C08961=1010.506,304.090,-163.238,-18.890,47.066,37.479
C08962=1010.613,303.852,-163.048,-19.485,46.587,36.235
C08963=1010.718,303.613,-162.860,-20.052,46.107,35.019
C08964=1010.823,303.374,-162.672,-20.593,45.627,33.826
C08965=1010.904,303.186,-162.527,-20.997,45.253,32.914
C08966=1010.984,302.998,-162.383,-21.384,44.880,32.017
C08967=1011.063,302.809,-162.239,-21.757,44.508,31.133
C08968=1011.142,302.619,-162.097,-22.115,44.137,30.264
C08969=1011.243,302.376,-161.916,-22.552,43.665,29.173
C08970=1011.342,302.132,-161.736,-22.967,43.196,28.105
C08971=1011.440,301.887,-161.558,-23.359,42.732,27.060
C08972=1011.536,301.641,-161.381,-23.731,42.271,26.037
C08973=1011.612,301.446,-161.243,-24.011,41.910,25.243
C08974=1011.687,301.252,-161.105,-24.278,41.553,24.463
C08975=1011.761,301.056,-160.968,-24.533,41.199,23.695
C08976=1011.835,300.859,-160.832,-24.778,40.847,22.938
C08977=1011.928,300.610,-160.662,-25.071,40.409,21.999
C08978=1012.020,300.361,-160.491,-25.349,39.974,21.077
C08979=1012.110,300.110,-160.323,-25.611,39.544,20.170
///RCONF 0,0,0,0,1,0,0,0,0,0,0,0,0,0,0,0,0,0,0,0,0,0,0,0
C08980=1012.200,299.859,-160.157,-25.857,39.121,19.283
C08981=1012.270,299.658,-160.024,-26.044,38.787,18.584
C08982=1012.340,299.456,-159.894,-26.221,38.458,17.898
C08983=1012.410,299.255,-159.763,-26.391,38.132,17.220
C08984=1012.478,299.051,-159.633,-26.551,37.810,16.553
C08985=1012.564,298.798,-159.472,-26.741,37.414,15.733
C08986=1012.647,298.543,-159.313,-26.918,37.024,14.926
C08987=1012.731,298.287,-159.155,-27.085,36.640,14.133
C08988=1012.814,298.031,-158.998,-27.241,36.263,13.354
C08989=1012.880,297.824,-158.872,-27.359,35.964,12.737
C08990=1012.944,297.618,-158.747,-27.470,35.670,12.129
C08991=1013.009,297.410,-158.624,-27.576,35.380,11.529
C08992=1013.072,297.202,-158.500,-27.675,35.094,10.935
C08993=1013.151,296.943,-158.349,-27.790,34.746,10.213
C08994=1013.228,296.685,-158.199,-27.897,34.404,9.500
C08995=1013.305,296.425,-158.050,-27.996,34.069,8.801
C08996=1013.380,296.164,-157.902,-28.087,33.740,8.111
C08997=1013.441,295.953,-157.783,-28.156,33.478,7.560
C08998=1013.502,295.741,-157.665,-28.220,33.220,7.016
C08999=1013.561,295.528,-157.547,-28.280,32.966,6.479
C09000=1013.621,295.315,-157.430,-28.335,32.716,5.947
C09001=1013.692,295.052,-157.288,-28.398,32.417,5.306
C09002=1013.763,294.790,-157.147,-28.455,32.123,4.674
C09003=1013.833,294.526,-157.006,-28.506,31.835,4.050
C09004=1013.902,294.263,-156.867,-28.552,31.552,3.436
C09005=1013.958,294.047,-156.754,-28.586,31.327,2.940
C09006=1014.014,293.830,-156.642,-28.617,31.104,2.450
C09007=1014.070,293.613,-156.531,-28.645,30.886,1.967
C09008=1014.124,293.395,-156.420,-28.669,30.673,1.490
C09009=1014.190,293.130,-156.286,-28.695,30.417,0.916
C09010=1014.254,292.865,-156.154,-28.717,30.168,0.353
C09011=1014.318,292.598,-156.022,-28.736,29.926,-0.203
C09012=1014.382,292.331,-155.891,-28.751,29.686,-0.753
C09013=1014.434,292.111,-155.784,-28.760,29.494,-1.200
C09014=1014.485,291.891,-155.678,-28.768,29.306,-1.642
C09015=1014.535,291.669,-155.572,-28.773,29.120,-2.080
C09016=1014.586,291.448,-155.467,-28.777,28.937,-2.514
C09017=1014.646,291.180,-155.341,-28.778,28.722,-3.030
C09018=1014.705,290.912,-155.217,-28.777,28.512,-3.541
C09019=1014.763,290.643,-155.093,-28.773,28.305,-4.046
C09020=1014.821,290.373,-154.970,-28.767,28.103,-4.544
C09021=1014.869,290.149,-154.869,-28.760,27.939,-4.952
C09022=1014.915,289.926,-154.768,-28.752,27.779,-5.357
C09023=1014.962,289.701,-154.668,-28.742,27.622,-5.757
C09024=1015.008,289.476,-154.569,-28.730,27.467,-6.153
C09025=1015.063,289.207,-154.450,-28.715,27.285,-6.624
C09026=1015.116,288.935,-154.333,-28.698,27.109,-7.088
C09027=1015.170,288.665,-154.217,-28.679,26.937,-7.545
C09028=1015.222,288.394,-154.102,-28.659,26.767,-7.999
C09029=1015.266,288.166,-154.006,-28.641,26.630,-8.372
C09030=1015.309,287.939,-153.911,-28.622,26.495,-8.743
C09031=1015.351,287.712,-153.816,-28.602,26.363,-9.109
C09032=1015.393,287.483,-153.722,-28.581,26.233,-9.471
C09033=1015.442,287.211,-153.611,-28.555,26.082,-9.899
C09034=1015.492,286.940,-153.500,-28.527,25.936,-10.320
C09035=1015.540,286.667,-153.391,-28.499,25.792,-10.737
C09036=1015.587,286.394,-153.283,-28.470,25.652,-11.148
C09037=1015.627,286.164,-153.192,-28.444,25.537,-11.492
C09038=1015.665,285.933,-153.102,-28.418,25.425,-11.832
C09039=1015.705,285.704,-153.012,-28.391,25.314,-12.171
C09040=1015.743,285.473,-152.924,-28.364,25.204,-12.507
C09041=1015.787,285.199,-152.820,-28.330,25.079,-12.901
C09042=1015.832,284.926,-152.716,-28.296,24.955,-13.292
C09043=1015.875,284.652,-152.614,-28.261,24.835,-13.680
C09044=1015.918,284.378,-152.512,-28.226,24.716,-14.065
C09045=1015.954,284.145,-152.426,-28.195,24.619,-14.388
C09046=1015.989,283.912,-152.341,-28.164,24.524,-14.708
C09047=1016.024,283.680,-152.256,-28.132,24.429,-15.026
C09048=1016.059,283.447,-152.172,-28.100,24.338,-15.343
C09049=1016.099,283.173,-152.075,-28.062,24.232,-15.713
C09050=1016.138,282.897,-151.978,-28.023,24.128,-16.079
C09051=1016.177,282.623,-151.881,-27.984,24.027,-16.441
C09052=1016.216,282.348,-151.786,-27.945,23.929,-16.801
C09053=1016.248,282.113,-151.705,-27.911,23.848,-17.104
C09054=1016.280,281.878,-151.625,-27.877,23.768,-17.406
C09055=1016.311,281.643,-151.545,-27.842,23.690,-17.706
C09056=1016.343,281.407,-151.466,-27.807,23.613,-18.004
C09057=1016.378,281.132,-151.374,-27.766,23.526,-18.349
C09058=1016.414,280.857,-151.284,-27.725,23.440,-18.691
C09059=1016.448,280.581,-151.193,-27.684,23.357,-19.031
C09060=1016.482,280.304,-151.104,-27.642,23.276,-19.367
C09061=1016.511,280.068,-151.028,-27.606,23.208,-19.653
C09062=1016.539,279.830,-150.952,-27.570,23.142,-19.936
C09063=1016.567,279.594,-150.877,-27.534,23.078,-20.218
C09064=1016.595,279.357,-150.803,-27.498,23.014,-20.499
C09065=1016.626,279.080,-150.717,-27.456,22.942,-20.824
C09066=1016.658,278.804,-150.632,-27.413,22.873,-21.147
C09067=1016.689,278.527,-150.548,-27.370,22.804,-21.469
C09068=1016.718,278.250,-150.465,-27.327,22.737,-21.789
C09069=1016.743,278.012,-150.393,-27.290,22.681,-22.062
C09070=1016.769,277.773,-150.322,-27.252,22.626,-22.334
C09071=1016.793,277.535,-150.252,-27.215,22.573,-22.606
C09072=1016.818,277.296,-150.183,-27.177,22.521,-22.877
C09073=1016.846,277.019,-150.102,-27.134,22.462,-23.186
C09074=1016.872,276.741,-150.023,-27.090,22.404,-23.496
C09075=1016.899,276.464,-149.944,-27.046,22.349,-23.804
C09076=1016.925,276.187,-149.866,-27.003,22.294,-24.111
C09077=1016.947,275.947,-149.800,-26.965,22.250,-24.373
C09078=1016.969,275.706,-149.733,-26.927,22.204,-24.635
C09079=1016.990,275.466,-149.667,-26.889,22.162,-24.896
C09080=1017.012,275.226,-149.602,-26.851,22.119,-25.156
C09081=1017.035,274.949,-149.528,-26.807,22.073,-25.453
C09082=1017.058,274.670,-149.454,-26.763,22.027,-25.750
C09083=1017.080,274.393,-149.380,-26.720,21.983,-26.043
C09084=1017.103,274.115,-149.308,-26.676,21.940,-26.336
C09085=1017.122,273.874,-149.246,-26.638,21.903,-26.590
C09086=1017.140,273.632,-149.184,-26.600,21.869,-26.841
C09087=1017.158,273.391,-149.123,-26.562,21.835,-27.092
C09088=1017.176,273.149,-149.062,-26.525,21.803,-27.342
C09089=1017.197,272.871,-148.993,-26.481,21.766,-27.626
C09090=1017.216,272.593,-148.925,-26.438,21.731,-27.910
C09091=1017.234,272.315,-148.857,-26.395,21.697,-28.194
C09092=1017.254,272.036,-148.790,-26.351,21.664,-28.476
C09093=1017.269,271.793,-148.732,-26.314,21.637,-28.720
C09094=1017.284,271.550,-148.675,-26.276,21.610,-28.964
C09095=1017.299,271.308,-148.618,-26.238,21.585,-29.208
C09096=1017.315,271.065,-148.561,-26.201,21.560,-29.450
C09097=1017.330,270.786,-148.498,-26.158,21.533,-29.728
C09098=1017.346,270.508,-148.435,-26.115,21.507,-30.003
C09099=1017.361,270.229,-148.372,-26.072,21.483,-30.277
C09100=1017.376,269.951,-148.310,-26.030,21.459,-30.551
C09101=1017.388,269.707,-148.257,-25.992,21.439,-30.791
C09102=1017.400,269.462,-148.204,-25.955,21.420,-31.029
C09103=1017.413,269.219,-148.151,-25.918,21.402,-31.266
C09104=1017.424,268.974,-148.098,-25.881,21.386,-31.502
C09105=1017.436,268.696,-148.040,-25.839,21.367,-31.772
C09106=1017.449,268.417,-147.983,-25.797,21.350,-32.039
C09107=1017.461,268.139,-147.926,-25.755,21.333,-32.307
C09108=1017.472,267.860,-147.869,-25.713,21.318,-32.573
C09109=1017.481,267.616,-147.820,-25.677,21.306,-32.805
C09110=1017.490,267.370,-147.771,-25.641,21.295,-33.037
C09111=1017.499,267.125,-147.723,-25.604,21.284,-33.269
C09112=1017.508,266.879,-147.676,-25.568,21.275,-33.499
C09113=1017.516,266.601,-147.622,-25.527,21.264,-33.760
C09114=1017.525,266.322,-147.569,-25.487,21.254,-34.021
C09115=1017.533,266.043,-147.517,-25.446,21.246,-34.279
C09116=1017.540,265.765,-147.465,-25.406,21.239,-34.538
C09117=1017.547,265.519,-147.421,-25.370,21.233,-34.766
C09118=1017.553,265.273,-147.376,-25.335,21.229,-34.991
C09119=1017.559,265.026,-147.333,-25.300,21.225,-35.219
C09120=1017.564,264.780,-147.290,-25.265,21.221,-35.444
C09121=1017.570,264.501,-147.242,-25.226,21.219,-35.699
C09122=1017.574,264.222,-147.194,-25.186,21.217,-35.952
C09123=1017.579,263.943,-147.146,-25.147,21.216,-36.205
C09124=1017.584,263.664,-147.100,-25.108,21.215,-36.458
C09125=1017.586,263.417,-147.059,-25.074,21.216,-36.681
C09126=1017.590,263.170,-147.020,-25.040,21.217,-36.903
C09127=1017.592,262.923,-146.980,-25.006,21.220,-37.124
C09128=1017.594,262.676,-146.941,-24.973,21.223,-37.345
C09129=1017.597,262.397,-146.898,-24.935,21.227,-37.593
C09130=1017.598,262.117,-146.855,-24.897,21.233,-37.842
C09131=1017.600,261.839,-146.813,-24.860,21.238,-38.090
C09132=1017.600,261.559,-146.771,-24.823,21.245,-38.337
C09133=1017.601,261.311,-146.736,-24.790,21.251,-38.554
C09134=1017.601,261.064,-146.700,-24.758,21.259,-38.770
C09135=1017.600,260.816,-146.665,-24.725,21.267,-38.988
C09136=1017.599,260.568,-146.631,-24.693,21.275,-39.204
C09137=1017.598,260.289,-146.592,-24.658,21.287,-39.446
C09138=1017.596,260.009,-146.554,-24.622,21.298,-39.688
C09139=1017.594,259.730,-146.517,-24.587,21.310,-39.930
C09140=1017.592,259.450,-146.481,-24.551,21.322,-40.171
C09141=1017.575,258.214,-146.327,-24.430,21.375,-41.012
C09142=1017.571,257.971,-146.298,-24.430,21.375,-41.014
C09143=1017.568,257.727,-146.269,-24.429,21.375,-41.018
C09144=1017.565,257.483,-146.240,-24.429,21.376,-41.019
C09145=1017.560,257.241,-146.210,-24.429,21.376,-41.021
C09146=1017.557,256.997,-146.181,-24.428,21.375,-41.025
C09147=1017.554,256.754,-146.152,-24.428,21.376,-41.027
C09148=1017.551,256.510,-146.123,-24.428,21.377,-41.029
C09149=1017.548,256.262,-146.094,-24.427,21.376,-41.032
C09150=1017.544,256.014,-146.063,-24.427,21.376,-41.034
C09151=1017.541,255.766,-146.035,-24.426,21.376,-41.037
C09152=1017.537,255.518,-146.005,-24.426,21.377,-41.040
C09153=1017.534,255.269,-145.975,-24.426,21.377,-41.042
C09154=1017.530,255.021,-145.945,-24.425,21.377,-41.045
C09155=1017.527,254.772,-145.916,-24.425,21.377,-41.047
C09156=1017.524,254.524,-145.887,-24.425,21.377,-41.049
C09157=1017.520,254.276,-145.856,-24.424,21.378,-41.052
C09158=1017.517,254.028,-145.828,-24.424,21.378,-41.054
C09159=1017.514,253.780,-145.797,-24.424,21.378,-41.058
C09160=1017.510,253.532,-145.768,-24.423,21.378,-41.060
C09161=1017.508,253.283,-145.739,-24.423,21.378,-41.061
C09162=1017.504,253.035,-145.709,-24.423,21.378,-41.065
C09163=1017.501,252.787,-145.680,-24.422,21.379,-41.067
C09164=1017.497,252.538,-145.651,-24.422,21.379,-41.069
C09165=1017.494,252.291,-145.621,-24.421,21.378,-41.072
C09166=1017.491,252.042,-145.591,-24.421,21.379,-41.074
C09167=1017.488,251.794,-145.562,-24.421,21.380,-41.076
C09168=1017.484,251.545,-145.533,-24.421,21.380,-41.078
C09169=1017.482,251.302,-145.504,-24.420,21.380,-41.082
C09170=1017.478,251.059,-145.475,-24.420,21.380,-41.084
C09171=1017.475,250.815,-145.446,-24.420,21.380,-41.085
C09172=1017.472,250.572,-145.417,-24.419,21.380,-41.089
C09173=1017.468,250.329,-145.389,-24.419,21.380,-41.091
C09174=1017.466,250.086,-145.360,-24.419,21.381,-41.093
C09175=1017.462,249.842,-145.332,-24.418,21.381,-41.095
C09176=1017.459,249.598,-145.303,-24.418,21.381,-41.098
C09177=1017.456,249.350,-145.274,-24.418,21.381,-41.100
C09178=1017.453,249.102,-145.244,-24.417,21.381,-41.102
C09179=1017.449,248.853,-145.215,-24.417,21.381,-41.104
C09180=1017.447,248.606,-145.185,-24.417,21.381,-41.107
C09181=1017.443,248.358,-145.156,-24.416,21.381,-41.109
C09182=1017.440,248.109,-145.127,-24.416,21.382,-41.111
C09183=1017.437,247.861,-145.098,-24.416,21.382,-41.113
C09184=1017.434,247.613,-145.069,-24.415,21.382,-41.117
C09185=1017.430,247.364,-145.039,-24.415,21.382,-41.118
C09186=1017.427,247.116,-145.011,-24.415,21.382,-41.120
C09187=1017.425,246.868,-144.981,-24.414,21.383,-41.122
C09188=1017.421,246.620,-144.952,-24.414,21.382,-41.126
C09189=1017.419,246.371,-144.923,-24.414,21.382,-41.127
C09190=1017.415,246.123,-144.894,-24.413,21.383,-41.129
C09191=1017.413,245.875,-144.865,-24.413,21.384,-41.132
C09192=1017.409,245.627,-144.836,-24.413,21.384,-41.134
C09193=1017.406,245.379,-144.807,-24.412,21.384,-41.137
C09194=1017.403,245.130,-144.777,-24.412,21.384,-41.139
C09195=1017.400,244.882,-144.748,-24.412,21.384,-41.141
C09196=1017.397,244.633,-144.719,-24.412,21.384,-41.143
C09197=1017.394,244.390,-144.692,-24.411,21.384,-41.144
C09198=1017.391,244.146,-144.662,-24.411,21.384,-41.148
C09199=1017.388,243.904,-144.634,-24.411,21.384,-41.150
C09200=1017.385,243.660,-144.606,-24.410,21.384,-41.151
C09201=1017.382,243.418,-144.578,-24.410,21.385,-41.153
C09202=1017.379,243.173,-144.549,-24.410,21.385,-41.155
C09203=1017.376,242.931,-144.521,-24.410,21.385,-41.157
C09204=1017.374,242.688,-144.492,-24.409,21.385,-41.159
C09205=1017.370,242.440,-144.463,-24.409,21.385,-41.162
C09206=1017.367,242.191,-144.435,-24.408,21.385,-41.164
C09207=1017.364,241.942,-144.405,-24.408,21.385,-41.166
C09208=1017.361,241.694,-144.377,-24.408,21.386,-41.168
C09209=1017.358,241.446,-144.347,-24.408,21.386,-41.170
C09210=1017.355,241.198,-144.319,-24.407,21.386,-41.172
C09211=1017.353,240.949,-144.290,-24.407,21.386,-41.174
C09212=1017.350,240.701,-144.261,-24.407,21.386,-41.177
C09213=1017.346,240.453,-144.232,-24.406,21.386,-41.179
C09214=1017.344,240.204,-144.204,-24.406,21.386,-41.181
C09215=1017.341,239.956,-144.175,-24.406,21.386,-41.183
C09216=1017.338,239.708,-144.145,-24.406,21.387,-41.184
C09217=1017.335,239.460,-144.117,-24.405,21.387,-41.186
C09218=1017.332,239.212,-144.089,-24.405,21.387,-41.188
C09219=1017.330,238.963,-144.059,-24.405,21.387,-41.190
C09220=1017.327,238.715,-144.031,-24.405,21.388,-41.192
C09221=1017.324,238.466,-144.002,-24.404,21.387,-41.195
C09222=1017.321,238.218,-143.974,-24.404,21.387,-41.197
C09223=1017.318,237.970,-143.945,-24.403,21.388,-41.199
C09224=1017.315,237.722,-143.916,-24.403,21.388,-41.201
C09225=1017.312,237.478,-143.888,-24.403,21.388,-41.203
C09226=1017.310,237.235,-143.859,-24.403,21.388,-41.205
C09227=1017.307,236.992,-143.832,-24.402,21.388,-41.207
C09228=1017.305,236.749,-143.803,-24.402,21.389,-41.209
C09229=1017.301,236.506,-143.775,-24.402,21.389,-41.210
C09230=1017.299,236.263,-143.748,-24.402,21.389,-41.212
C09231=1017.296,236.019,-143.719,-24.401,21.389,-41.214
C09232=1017.293,235.777,-143.691,-24.401,21.390,-41.216
C09233=1017.291,235.528,-143.662,-24.401,21.389,-41.218
C09234=1017.288,235.280,-143.634,-24.401,21.389,-41.219
C09235=1017.285,235.031,-143.606,-24.400,21.389,-41.221
C09236=1017.283,234.784,-143.577,-24.400,21.390,-41.223
C09237=1017.280,234.535,-143.549,-24.400,21.390,-41.225
C09238=1017.277,234.287,-143.519,-24.400,21.390,-41.227
C09239=1017.274,234.038,-143.491,-24.399,21.390,-41.229
C09240=1017.271,233.790,-143.463,-24.399,21.390,-41.231
C09241=1017.269,233.541,-143.434,-24.399,21.391,-41.233
C09242=1017.266,233.293,-143.406,-24.399,21.391,-41.234
C09243=1017.264,233.045,-143.377,-24.398,21.391,-41.236
C09244=1017.261,232.797,-143.349,-24.398,21.390,-41.238
C09245=1017.258,232.548,-143.320,-24.398,21.391,-41.240
C09246=1017.255,232.300,-143.291,-24.397,21.391,-41.242
C09247=1017.252,232.051,-143.263,-24.397,21.391,-41.243
C09248=1017.249,231.803,-143.234,-24.397,21.391,-41.245
C09249=1017.248,231.555,-143.206,-24.397,21.392,-41.247
C09250=1017.245,231.306,-143.178,-24.396,21.392,-41.249
C09251=1017.242,231.057,-143.149,-24.396,21.392,-41.251
C09252=1017.239,230.809,-143.120,-24.396,21.391,-41.252
C09253=1017.237,230.587,-143.095,-24.396,21.392,-41.254
C09254=1017.235,230.365,-143.071,-24.395,21.392,-41.256
C09255=1017.233,230.143,-143.045,-24.395,21.392,-41.258
C09256=1017.230,229.920,-143.020,-24.395,21.392,-41.258
C09257=1017.228,229.698,-142.994,-24.395,21.392,-41.260
C09258=1017.225,229.476,-142.969,-24.395,21.392,-41.262
C09259=1017.223,229.254,-142.943,-24.394,21.393,-41.264
C09260=1017.221,229.031,-142.917,-24.394,21.392,-41.265
C09261=1017.218,228.783,-142.889,-24.394,21.392,-41.267
C09262=1017.216,228.535,-142.862,-24.394,21.392,-41.269
C09263=1017.214,228.286,-142.833,-24.393,21.393,-41.271
C09264=1017.210,228.038,-142.804,-24.393,21.393,-41.273
C09265=1017.209,227.790,-142.776,-24.393,21.394,-41.273
C09266=1017.206,227.541,-142.748,-24.393,21.393,-41.275
C09267=1017.203,227.292,-142.720,-24.393,21.393,-41.276
C09268=1017.201,227.044,-142.691,-24.392,21.394,-41.278
C09269=1017.198,226.796,-142.663,-24.392,21.394,-41.280
C09270=1017.195,226.548,-142.635,-24.392,21.394,-41.282
C09271=1017.193,226.299,-142.606,-24.392,21.394,-41.284
C09272=1017.190,226.051,-142.578,-24.391,21.394,-41.285
C09273=1017.188,225.802,-142.550,-24.391,21.394,-41.287
C09274=1017.186,225.554,-142.522,-24.391,21.394,-41.289
C09275=1017.183,225.305,-142.494,-24.390,21.394,-41.291
C09276=1017.181,225.057,-142.465,-24.391,21.395,-41.291
C09277=1017.179,224.767,-142.433,-24.390,21.395,-41.293
C09278=1017.176,224.478,-142.400,-24.390,21.395,-41.295
C09279=1017.172,224.188,-142.367,-24.389,21.394,-41.298
C09280=1017.169,223.898,-142.335,-24.389,21.395,-41.300
C09281=1017.167,223.655,-142.306,-24.389,21.395,-41.300
C09282=1017.165,223.412,-142.279,-24.389,21.396,-41.302
C09283=1017.162,223.170,-142.252,-24.389,21.396,-41.304
C09284=1017.160,222.926,-142.224,-24.388,21.395,-41.306
C09285=1017.158,222.684,-142.197,-24.388,21.395,-41.308
C09286=1017.155,222.441,-142.170,-24.388,21.396,-41.309
C09287=1017.153,222.198,-142.141,-24.388,21.397,-41.310
C09288=1017.151,221.955,-142.114,-24.388,21.396,-41.311
C09289=1017.148,221.706,-142.086,-24.387,21.396,-41.313
C09290=1017.146,221.458,-142.058,-24.387,21.396,-41.315
C09291=1017.143,221.210,-142.030,-24.387,21.397,-41.317
C09292=1017.141,220.961,-142.003,-24.386,21.396,-41.318
C09293=1017.139,220.712,-141.974,-24.386,21.396,-41.320
C09294=1017.137,220.464,-141.946,-24.386,21.397,-41.321
C09295=1017.134,220.216,-141.918,-24.386,21.397,-41.323
C09296=1017.132,219.968,-141.890,-24.386,21.397,-41.324
C09297=1017.130,219.720,-141.862,-24.385,21.397,-41.326
C09298=1017.128,219.471,-141.834,-24.385,21.397,-41.328
C09299=1017.125,219.222,-141.807,-24.385,21.397,-41.330
C09300=1017.123,218.974,-141.779,-24.385,21.397,-41.330
C09301=1017.121,218.725,-141.750,-24.385,21.397,-41.332
C09302=1017.118,218.477,-141.722,-24.384,21.398,-41.333
C09303=1017.116,218.229,-141.695,-24.384,21.398,-41.335
C09304=1017.114,217.980,-141.667,-24.384,21.397,-41.337
C09305=1017.111,217.732,-141.639,-24.384,21.397,-41.339
C09306=1017.110,217.483,-141.611,-24.384,21.398,-41.339
C09307=1017.107,217.236,-141.583,-24.383,21.399,-41.341
C09308=1017.105,216.986,-141.556,-24.383,21.398,-41.342
C09309=1017.102,216.744,-141.528,-24.383,21.398,-41.344
C09310=1017.101,216.501,-141.501,-24.383,21.398,-41.346
C09311=1017.098,216.258,-141.473,-24.383,21.398,-41.346
C09312=1017.096,216.015,-141.447,-24.382,21.399,-41.348
C09313=1017.094,215.773,-141.420,-24.382,21.399,-41.350
C09314=1017.092,215.530,-141.392,-24.382,21.399,-41.352
C09315=1017.090,215.287,-141.365,-24.382,21.398,-41.353
C09316=1017.088,215.045,-141.338,-24.382,21.399,-41.354
C09317=1017.086,214.795,-141.310,-24.381,21.400,-41.356
C09318=1017.083,214.547,-141.282,-24.381,21.399,-41.357
C09319=1017.081,214.299,-141.255,-24.381,21.399,-41.359
C09320=1017.080,214.051,-141.227,-24.381,21.400,-41.359
C09321=1017.077,213.802,-141.199,-24.381,21.400,-41.361
C09322=1017.075,213.554,-141.172,-24.380,21.400,-41.363
C09323=1017.073,213.305,-141.143,-24.380,21.400,-41.365
C09324=1017.071,213.057,-141.116,-24.380,21.400,-41.366
C09325=1017.069,212.808,-141.088,-24.380,21.400,-41.366
C09326=1017.066,212.560,-141.060,-24.380,21.400,-41.368
C09327=1017.064,212.312,-141.033,-24.379,21.400,-41.370
C09328=1017.063,212.063,-141.005,-24.379,21.400,-41.372
C09329=1017.060,211.814,-140.977,-24.379,21.401,-41.372
C09330=1017.058,211.566,-140.950,-24.379,21.401,-41.374
C09331=1017.056,211.318,-140.922,-24.378,21.400,-41.375
C09332=1017.054,211.070,-140.894,-24.378,21.400,-41.377
C09333=1017.052,210.820,-140.866,-24.378,21.401,-41.378
C09334=1017.050,210.572,-140.839,-24.378,21.401,-41.379
C09335=1017.048,210.324,-140.812,-24.378,21.401,-41.381
C09336=1017.046,210.076,-140.783,-24.377,21.401,-41.383
C09337=1017.044,209.832,-140.757,-24.377,21.401,-41.383
C09338=1017.042,209.590,-140.730,-24.377,21.401,-41.385
C09339=1017.040,209.348,-140.703,-24.377,21.402,-41.387
C09340=1017.038,209.105,-140.677,-24.377,21.401,-41.388
C09341=1017.036,208.862,-140.649,-24.377,21.402,-41.389
C09342=1017.034,208.619,-140.622,-24.376,21.402,-41.391
C09343=1017.032,208.377,-140.595,-24.376,21.401,-41.392
C09344=1017.030,208.134,-140.569,-24.376,21.402,-41.392
C09345=1017.029,207.886,-140.541,-24.376,21.402,-41.394
C09346=1017.027,207.637,-140.514,-24.376,21.402,-41.396
C09347=1017.024,207.389,-140.486,-24.375,21.402,-41.398
C09348=1017.022,207.140,-140.458,-24.375,21.402,-41.398
C09349=1017.020,206.891,-140.431,-24.375,21.402,-41.399
C09350=1017.019,206.643,-140.403,-24.375,21.402,-41.401
C09351=1017.017,206.395,-140.376,-24.375,21.402,-41.401
C09352=1017.015,206.146,-140.349,-24.375,21.403,-41.403
C09353=1017.013,205.898,-140.321,-24.374,21.403,-41.405
C09354=1017.011,205.649,-140.294,-24.374,21.402,-41.407
C09355=1017.009,205.401,-140.267,-24.374,21.403,-41.407
C09356=1017.007,205.153,-140.238,-24.374,21.403,-41.409
C09357=1017.005,204.904,-140.211,-24.373,21.403,-41.410
C09358=1017.004,204.655,-140.184,-24.374,21.404,-41.411
C09359=1017.002,204.407,-140.157,-24.373,21.403,-41.412
C09360=1017.000,204.159,-140.129,-24.373,21.403,-41.414
C09361=1016.998,203.910,-140.101,-24.373,21.404,-41.415
C09362=1016.996,203.662,-140.074,-24.373,21.403,-41.416
C09363=1016.990,202.446,-139.939,-24.425,21.378,-41.051
C09364=1016.989,202.057,-139.895,-24.424,21.378,-41.052
C09365=1016.989,201.709,-139.856,-24.424,21.378,-41.054
C09366=1016.989,201.358,-139.818,-24.424,21.378,-41.058
C09367=1016.990,200.950,-139.773,-24.423,21.379,-41.060
C09368=1016.991,200.722,-139.748,-24.423,21.378,-41.061
C09369=1016.991,200.494,-139.723,-24.423,21.378,-41.063
C09370=1016.991,200.271,-139.699,-24.423,21.378,-41.065
C09371=1016.992,200.058,-139.675,-24.423,21.378,-41.065
C09372=1016.992,199.658,-139.631,-24.422,21.379,-41.069
C09373=1016.992,199.269,-139.589,-24.422,21.379,-41.071
C09374=1016.994,198.870,-139.545,-24.421,21.379,-41.074
C09375=1016.994,198.469,-139.502,-24.421,21.379,-41.076
C09376=1016.995,198.068,-139.458,-24.421,21.380,-41.078
C09377=1016.995,197.666,-139.414,-24.420,21.380,-41.082
C09378=1016.996,197.266,-139.369,-24.420,21.380,-41.084
C09379=1016.997,196.864,-139.326,-24.419,21.380,-41.087
C09380=1016.998,196.463,-139.283,-24.419,21.380,-41.089
C09381=1016.998,196.062,-139.239,-24.419,21.381,-41.091
C09382=1016.999,195.661,-139.195,-24.418,21.380,-41.094
C09383=1017.000,195.260,-139.151,-24.418,21.381,-41.097
C09384=1017.001,194.859,-139.107,-24.418,21.381,-41.100
C09385=1017.002,194.458,-139.064,-24.417,21.381,-41.102
C09386=1017.002,194.057,-139.021,-24.417,21.381,-41.105
C09387=1017.003,193.656,-138.977,-24.417,21.382,-41.108
C09388=1017.004,193.255,-138.933,-24.416,21.382,-41.109
C09389=1017.005,192.853,-138.889,-24.416,21.382,-41.113
C09390=1017.006,192.452,-138.846,-24.415,21.382,-41.115
C09391=1017.006,192.051,-138.803,-24.415,21.382,-41.118
C09392=1017.007,191.650,-138.760,-24.415,21.382,-41.120
C09393=1017.008,191.249,-138.716,-24.414,21.382,-41.124
C09394=1017.009,190.848,-138.672,-24.414,21.383,-41.126
C09395=1017.010,190.446,-138.628,-24.414,21.383,-41.128
C09396=1017.011,190.046,-138.585,-24.413,21.383,-41.131
C09397=1017.012,189.645,-138.542,-24.413,21.383,-41.133
C09398=1017.013,189.243,-138.499,-24.412,21.384,-41.137
C09399=1017.013,188.842,-138.455,-24.412,21.384,-41.139
C09400=1017.014,188.441,-138.412,-24.412,21.384,-41.141
C09401=1017.016,188.041,-138.369,-24.411,21.384,-41.144
C09402=1017.016,187.639,-138.326,-24.411,21.385,-41.146
C09403=1017.018,187.238,-138.282,-24.411,21.384,-41.150
C09404=1017.019,186.837,-138.239,-24.410,21.384,-41.151
C09405=1017.020,186.436,-138.196,-24.410,21.384,-41.155
C09406=1017.021,186.035,-138.152,-24.410,21.385,-41.157
C09407=1017.022,185.634,-138.109,-24.409,21.385,-41.159
C09408=1017.023,185.233,-138.066,-24.409,21.385,-41.162
C09409=1017.024,184.832,-138.023,-24.409,21.386,-41.165
C09410=1017.025,184.431,-137.980,-24.408,21.386,-41.168
C09411=1017.026,184.030,-137.936,-24.408,21.386,-41.170
C09412=1017.027,183.630,-137.894,-24.407,21.386,-41.172
C09413=1017.028,183.228,-137.850,-24.407,21.386,-41.176
C09414=1017.029,182.828,-137.807,-24.407,21.387,-41.177
C09415=1017.030,182.426,-137.765,-24.406,21.386,-41.181
C09416=1017.031,182.026,-137.722,-24.406,21.387,-41.183
C09417=1017.032,181.624,-137.678,-24.405,21.387,-41.186
C09418=1017.034,181.224,-137.635,-24.405,21.387,-41.188
C09419=1017.034,180.824,-137.593,-24.405,21.387,-41.190
C09420=1017.035,180.422,-137.551,-24.404,21.388,-41.194
C09421=1017.037,180.021,-137.508,-24.404,21.388,-41.196
C09422=1017.038,179.621,-137.465,-24.403,21.388,-41.199
C09423=1017.039,179.220,-137.421,-24.403,21.388,-41.201
C09424=1017.040,178.819,-137.378,-24.403,21.388,-41.205
C09425=1017.042,178.418,-137.336,-24.402,21.388,-41.207
C09426=1017.042,178.017,-137.293,-24.402,21.389,-41.209
C09427=1017.044,177.616,-137.250,-24.402,21.389,-41.212
C09428=1017.044,177.216,-137.208,-24.401,21.389,-41.214
C09429=1017.046,176.815,-137.165,-24.401,21.389,-41.218
C09430=1017.047,176.414,-137.122,-24.401,21.389,-41.219
C09431=1017.048,176.013,-137.079,-24.400,21.390,-41.223
C09432=1017.050,175.612,-137.037,-24.400,21.390,-41.225
C09433=1017.050,175.212,-136.994,-24.400,21.390,-41.227
C09434=1017.052,174.811,-136.951,-24.399,21.390,-41.231
C09435=1017.053,174.410,-136.909,-24.399,21.391,-41.233
C09436=1017.055,174.010,-136.866,-24.398,21.390,-41.236
C09437=1017.055,173.610,-136.824,-24.398,21.390,-41.238
C09438=1017.057,173.208,-136.782,-24.397,21.391,-41.242
C09439=1017.058,172.808,-136.739,-24.397,21.391,-41.243
C09440=1017.060,172.407,-136.696,-24.397,21.391,-41.247
C09441=1017.061,172.007,-136.654,-24.396,21.392,-41.249
C09442=1017.062,171.606,-136.611,-24.396,21.392,-41.251
C09443=1017.064,171.205,-136.569,-24.396,21.392,-41.254
C09444=1017.064,170.805,-136.527,-24.395,21.392,-41.256
C09445=1017.066,170.405,-136.484,-24.395,21.392,-41.260
C09446=1017.068,170.004,-136.442,-24.395,21.392,-41.262
C09447=1017.068,169.604,-136.399,-24.394,21.392,-41.265
C09448=1017.070,169.203,-136.357,-24.394,21.393,-41.267
C09449=1017.071,168.802,-136.315,-24.393,21.393,-41.271
C09450=1017.073,168.403,-136.272,-24.393,21.393,-41.273
C09451=1017.074,168.001,-136.230,-24.393,21.394,-41.275
C09452=1017.075,167.601,-136.188,-24.392,21.394,-41.278
C09453=1017.077,167.200,-136.146,-24.392,21.394,-41.280
C09454=1017.078,166.801,-136.104,-24.391,21.393,-41.284
C09455=1017.079,166.400,-136.061,-24.391,21.395,-41.286
C09456=1017.081,166.000,-136.019,-24.391,21.394,-41.289
C09457=1017.082,165.599,-135.977,-24.390,21.394,-41.291
C09458=1017.083,165.199,-135.935,-24.390,21.395,-41.295
C09459=1017.085,164.798,-135.893,-24.390,21.395,-41.297
C09460=1017.086,164.398,-135.850,-24.389,21.395,-41.300
C09461=1017.088,164.012,-135.811,-24.389,21.395,-41.302
C09462=1017.088,163.822,-135.790,-24.389,21.395,-41.304
C09463=1017.089,163.410,-135.747,-24.388,21.396,-41.306
C09464=1017.090,163.175,-135.722,-24.388,21.395,-41.308
C09465=1017.091,162.921,-135.696,-24.388,21.396,-41.309
C09466=1017.092,162.658,-135.667,-24.388,21.396,-41.311
C09467=1017.093,162.389,-135.640,-24.387,21.396,-41.313
C09468=1017.094,162.118,-135.611,-24.387,21.396,-41.315
C09469=1017.095,161.849,-135.583,-24.387,21.397,-41.317
C09470=1017.096,161.585,-135.556,-24.387,21.397,-41.319
C09471=1017.097,161.336,-135.529,-24.386,21.396,-41.320
C09472=1017.098,161.098,-135.504,-24.386,21.396,-41.322
C09473=1017.098,160.873,-135.481,-24.386,21.397,-41.324
C09474=1017.099,160.661,-135.459,-24.386,21.397,-41.325
C09475=1017.101,160.255,-135.416,-24.385,21.397,-41.328
C09476=1017.102,159.858,-135.374,-24.385,21.397,-41.330
C09477=1017.106,159.457,-135.334,-24.384,21.398,-41.333
C09478=1017.112,159.058,-135.295,-24.384,21.398,-41.335
C09479=1017.119,158.656,-135.256,-24.384,21.397,-41.339
C09480=1017.126,158.254,-135.218,-24.383,21.399,-41.341
C09481=1017.132,157.851,-135.179,-24.383,21.398,-41.344
C09482=1017.138,157.448,-135.140,-24.383,21.398,-41.346
C09483=1017.145,157.043,-135.101,-24.382,21.399,-41.350
C09484=1017.152,156.639,-135.062,-24.382,21.399,-41.352
C09485=1017.158,156.232,-135.023,-24.381,21.399,-41.355
C09486=1017.165,155.826,-134.983,-24.381,21.400,-41.358
C09487=1017.172,155.419,-134.944,-24.381,21.399,-41.361
C09488=1017.178,155.009,-134.905,-24.380,21.400,-41.363
C09489=1017.185,154.601,-134.865,-24.380,21.400,-41.366
C09490=1017.191,154.191,-134.826,-24.380,21.400,-41.368
C09491=1017.197,153.780,-134.786,-24.379,21.401,-41.372
C09492=1017.204,153.369,-134.746,-24.378,21.400,-41.375
C09493=1017.210,152.957,-134.707,-24.378,21.400,-41.377
C09494=1017.217,152.545,-134.666,-24.378,21.401,-41.381
C09495=1017.224,152.132,-134.628,-24.377,21.401,-41.383
C09496=1017.230,151.720,-134.587,-24.377,21.402,-41.387
C09497=1017.236,151.306,-134.547,-24.377,21.402,-41.389
C09498=1017.243,150.893,-134.508,-24.376,21.401,-41.392
C09499=1017.249,150.478,-134.467,-24.376,21.402,-41.394
C09500=1017.256,150.065,-134.427,-24.375,21.402,-41.398
C09501=1017.263,149.651,-134.388,-24.375,21.402,-41.401
C09502=1017.268,149.236,-134.348,-24.375,21.403,-41.403
C09503=1017.275,148.823,-134.308,-24.374,21.403,-41.407
C09504=1017.281,148.409,-134.268,-24.374,21.403,-41.409
C09505=1017.287,147.995,-134.228,-24.373,21.403,-41.412
C09506=1017.293,147.580,-134.189,-24.373,21.403,-41.416
C09507=1017.300,147.167,-134.149,-24.372,21.404,-41.418
C09508=1017.306,146.754,-134.109,-24.372,21.404,-41.422
C09509=1017.313,146.340,-134.069,-24.372,21.404,-41.424
C09510=1017.318,145.927,-134.030,-24.371,21.405,-41.427
C09511=1017.325,145.515,-133.990,-24.371,21.404,-41.431
C09512=1017.331,145.103,-133.950,-24.370,21.405,-41.432
C09513=1017.337,144.692,-133.910,-24.370,21.405,-41.436
C09514=1017.343,144.280,-133.870,-24.370,21.405,-41.438
C09515=1017.349,143.871,-133.831,-24.369,21.406,-41.442
C09516=1017.355,143.461,-133.792,-24.369,21.405,-41.445
C09517=1017.361,143.053,-133.753,-24.368,21.406,-41.448
C09518=1017.367,142.644,-133.713,-24.368,21.406,-41.451
C09519=1017.373,142.237,-133.674,-24.368,21.406,-41.453
C09520=1017.379,141.831,-133.635,-24.367,21.407,-41.457
C09521=1017.385,141.426,-133.596,-24.366,21.406,-41.460
C09522=1017.391,141.021,-133.557,-24.366,21.407,-41.462
C09523=1017.397,140.604,-133.517,-24.366,21.408,-41.466
C09524=1017.400,140.368,-133.495,-24.366,21.408,-41.468
C09525=1017.404,140.109,-133.470,-24.365,21.408,-41.470
C09526=1017.408,139.832,-133.443,-24.365,21.408,-41.471
C09527=1017.412,139.544,-133.416,-24.365,21.408,-41.473
C09528=1017.416,139.256,-133.388,-24.364,21.408,-41.475
C09529=1017.420,138.979,-133.361,-24.364,21.407,-41.476
C09530=1017.423,138.719,-133.337,-24.364,21.408,-41.478
C09531=1017.427,138.482,-133.314,-24.364,21.408,-41.480
C09532=1017.430,138.265,-133.293,-24.363,21.408,-41.482
C09533=1017.433,138.059,-133.273,-24.363,21.408,-41.484
C09534=1017.439,137.658,-133.234,-24.363,21.408,-41.486
C09535=1017.445,137.288,-133.199,-24.363,21.410,-41.488
C09536=1017.449,136.951,-133.167,-24.362,21.409,-41.491
C09537=1017.453,136.635,-133.136,-24.361,21.409,-41.495
C09538=1017.458,136.317,-133.106,-24.361,21.410,-41.497
C09539=1017.462,135.978,-133.073,-24.361,21.409,-41.500
C09540=1017.468,135.606,-133.038,-24.360,21.410,-41.502
C09541=1017.473,135.211,-133.000,-24.360,21.411,-41.505
C09542=1017.478,134.812,-132.962,-24.360,21.410,-41.508
C09543=1017.484,134.414,-132.923,-24.359,21.411,-41.510
C09544=1017.490,134.014,-132.885,-24.359,21.411,-41.514
C09545=1017.495,133.617,-132.847,-24.358,21.411,-41.517
C09546=1017.500,133.217,-132.809,-24.358,21.412,-41.519
C09547=1017.506,132.819,-132.771,-24.358,21.411,-41.523
C09548=1017.511,132.420,-132.732,-24.357,21.412,-41.525
C09549=1017.517,132.021,-132.695,-24.357,21.412,-41.528
C09550=1017.522,131.623,-132.656,-24.356,21.412,-41.532
C09551=1017.528,131.224,-132.618,-24.356,21.413,-41.534
C09552=1017.533,130.825,-132.580,-24.356,21.413,-41.538
C09553=1017.539,130.427,-132.542,-24.355,21.413,-41.541
C09554=1017.543,130.028,-132.504,-24.355,21.413,-41.543
C09555=1017.549,129.629,-132.466,-24.354,21.413,-41.547
C09556=1017.554,129.231,-132.427,-24.354,21.413,-41.550
C09557=1017.560,128.832,-132.390,-24.354,21.414,-41.552
C09558=1017.565,128.434,-132.351,-24.353,21.414,-41.555
C09559=1017.570,128.036,-132.313,-24.353,21.415,-41.558
C09560=1017.575,127.636,-132.275,-24.352,21.414,-41.561
C09561=1017.581,127.239,-132.237,-24.352,21.415,-41.565
C09562=1017.585,126.839,-132.199,-24.351,21.415,-41.567
C09563=1017.591,126.441,-132.160,-24.351,21.415,-41.571
C09564=1017.596,126.042,-132.123,-24.350,21.415,-41.574
C09565=1017.601,125.644,-132.085,-24.350,21.416,-41.576
C09566=1017.607,125.245,-132.047,-24.350,21.416,-41.580
C09567=1017.611,124.846,-132.008,-24.349,21.416,-41.583
C09568=1017.617,124.448,-131.971,-24.349,21.416,-41.585
C09569=1017.621,124.049,-131.933,-24.348,21.417,-41.589
C09570=1017.627,123.651,-131.895,-24.348,21.416,-41.592
C09571=1017.632,123.252,-131.856,-24.348,21.418,-41.595
C09572=1017.636,122.854,-131.818,-24.347,21.417,-41.598
C09573=1017.642,122.455,-131.781,-24.347,21.418,-41.602
C09574=1017.646,122.057,-131.742,-24.346,21.417,-41.605
C09575=1017.652,121.658,-131.705,-24.346,21.418,-41.607
C09576=1017.656,121.260,-131.667,-24.345,21.418,-41.611
C09577=1017.662,120.861,-131.629,-24.345,21.418,-41.614
C09578=1017.666,120.463,-131.591,-24.345,21.419,-41.617
C09579=1017.672,120.064,-131.554,-24.344,21.419,-41.620
C09580=1017.677,119.666,-131.515,-24.343,21.419,-41.624
C09581=1017.682,119.267,-131.478,-24.343,21.420,-41.626
C09582=1017.688,118.869,-131.440,-24.343,21.420,-41.629
C09583=1017.693,118.470,-131.403,-24.342,21.420,-41.633
C09584=1017.698,118.072,-131.365,-24.342,21.420,-41.637
C09585=1017.703,117.673,-131.327,-24.341,21.420,-41.638
C09586=1017.708,117.274,-131.290,-24.341,21.421,-41.642
C09587=1017.713,116.876,-131.252,-24.340,21.420,-41.646
C09588=1017.719,116.478,-131.214,-24.340,21.421,-41.649
C09589=1017.724,116.079,-131.177,-24.340,21.422,-41.652
C09590=1017.729,115.680,-131.139,-24.339,21.422,-41.655
C09591=1017.734,115.283,-131.101,-24.339,21.422,-41.659
C09592=1017.739,114.884,-131.064,-24.338,21.422,-41.662
C09593=1017.744,114.485,-131.026,-24.338,21.423,-41.664
C09594=1017.749,114.087,-130.988,-24.337,21.422,-41.668
C09595=1017.754,113.688,-130.951,-24.337,21.423,-41.671
C09596=1017.760,113.290,-130.913,-24.336,21.423,-41.675
C09597=1017.765,112.891,-130.876,-24.336,21.423,-41.677
C09598=1017.769,112.493,-130.838,-24.335,21.424,-41.681
C09599=1017.774,112.094,-130.801,-24.335,21.423,-41.684
C09600=1017.779,111.696,-130.763,-24.334,21.424,-41.688
C09601=1017.784,111.296,-130.726,-24.334,21.425,-41.690
C09602=1017.789,110.899,-130.688,-24.334,21.425,-41.694
C09603=1017.793,110.500,-130.651,-24.333,21.425,-41.697
C09604=1017.799,110.101,-130.613,-24.333,21.425,-41.701
C09605=1017.804,109.702,-130.576,-24.332,21.426,-41.703
C09606=1017.809,109.304,-130.538,-24.332,21.426,-41.707
C09607=1017.813,108.906,-130.501,-24.331,21.426,-41.710
C09608=1017.818,108.507,-130.463,-24.331,21.426,-41.714
C09609=1017.823,108.108,-130.426,-24.330,21.426,-41.717
C09610=1017.828,107.710,-130.388,-24.330,21.427,-41.719
C09611=1017.832,107.311,-130.351,-24.330,21.427,-41.723
C09612=1017.837,106.912,-130.313,-24.329,21.427,-41.727
C09613=1017.842,106.514,-130.276,-24.328,21.427,-41.730
C09614=1017.847,106.115,-130.239,-24.328,21.428,-41.734
C09615=1017.852,105.717,-130.201,-24.328,21.428,-41.736
C09616=1017.856,105.318,-130.164,-24.327,21.429,-41.740
C09617=1017.861,104.919,-130.126,-24.327,21.429,-41.743
C09618=1017.865,104.521,-130.089,-24.326,21.429,-41.747
C09619=1017.870,104.122,-130.052,-24.326,21.429,-41.751
C09620=1017.875,103.723,-130.014,-24.325,21.430,-41.754
C09621=1017.879,103.325,-129.976,-24.325,21.430,-41.756
C09622=1017.884,102.926,-129.939,-24.324,21.430,-41.760
C09623=1017.888,102.527,-129.902,-24.324,21.430,-41.763
C09624=1017.893,102.128,-129.864,-24.323,21.430,-41.767
C09625=1017.897,101.729,-129.827,-24.323,21.431,-41.771
C09626=1017.903,101.331,-129.790,-24.322,21.431,-41.775
C09627=1017.907,100.932,-129.753,-24.322,21.431,-41.778
C09628=1017.911,100.533,-129.716,-24.322,21.432,-41.780
C09629=1017.916,100.134,-129.678,-24.321,21.432,-41.784
C09630=1017.920,99.736,-129.640,-24.320,21.432,-41.787
C09631=1017.925,99.338,-129.603,-24.320,21.432,-41.791
C09632=1017.929,98.939,-129.566,-24.319,21.433,-41.795
C09633=1017.933,98.540,-129.529,-24.319,21.432,-41.798
C09634=1017.938,98.141,-129.491,-24.318,21.433,-41.802
C09635=1017.942,97.742,-129.454,-24.318,21.433,-41.806
C09636=1017.947,97.343,-129.416,-24.318,21.434,-41.808
C09637=1017.951,96.944,-129.379,-24.317,21.434,-41.811
C09638=1017.955,96.545,-129.342,-24.317,21.435,-41.815
C09639=1017.959,96.146,-129.305,-24.316,21.435,-41.819
C09640=1017.964,95.747,-129.268,-24.316,21.435,-41.822
C09641=1017.968,95.348,-129.230,-24.315,21.435,-41.826
C09642=1017.972,94.950,-129.193,-24.315,21.436,-41.830
C09643=1017.977,94.550,-129.156,-24.314,21.435,-41.833
C09644=1017.982,94.151,-129.119,-24.313,21.436,-41.837
C09645=1017.986,93.752,-129.082,-24.313,21.436,-41.841
C09646=1017.990,93.353,-129.045,-24.312,21.437,-41.844
C09647=1017.995,92.954,-129.008,-24.312,21.437,-41.846
C09648=1017.998,92.555,-128.970,-24.312,21.437,-41.850
C09649=1018.002,92.156,-128.933,-24.311,21.438,-41.854
C09650=1018.006,91.757,-128.896,-24.311,21.438,-41.857
C09651=1018.010,91.358,-128.859,-24.310,21.438,-41.861
C09652=1018.015,90.959,-128.823,-24.310,21.438,-41.865
C09653=1018.019,90.559,-128.785,-24.309,21.439,-41.868
C09654=1018.023,90.160,-128.748,-24.309,21.439,-41.872
C09655=1018.027,89.762,-128.711,-24.308,21.439,-41.875
C09656=1018.031,89.369,-128.674,-24.308,21.439,-41.879
C09657=1018.035,88.983,-128.638,-24.307,21.440,-41.883
C09658=1018.039,88.600,-128.603,-24.307,21.440,-41.887
C09659=1018.042,88.216,-128.568,-24.306,21.440,-41.890
C09660=1018.046,87.828,-128.532,-24.305,21.440,-41.894
C09661=1018.050,87.432,-128.494,-24.305,21.441,-41.898
C09662=1018.055,87.029,-128.457,-24.304,21.441,-41.901
C09663=1018.059,86.624,-128.419,-24.304,21.442,-41.905
C09664=1018.062,86.216,-128.381,-24.303,21.441,-41.908
C09665=1018.067,85.807,-128.344,-24.303,21.442,-41.912
C09666=1018.071,85.396,-128.306,-24.302,21.442,-41.916
C09667=1018.075,84.984,-128.268,-24.302,21.443,-41.920
C09668=1018.079,84.569,-128.229,-24.301,21.443,-41.923
C09669=1018.083,84.153,-128.190,-24.301,21.443,-41.927
C09670=1018.087,83.737,-128.152,-24.300,21.444,-41.931
C09671=1018.091,83.317,-128.113,-24.300,21.444,-41.935
C09672=1018.095,82.897,-128.074,-24.299,21.444,-41.938
C09673=1018.097,82.687,-128.055,-24.299,21.444,-41.940
C09674=1018.099,82.476,-128.036,-24.299,21.444,-41.942
C09675=1018.101,82.265,-128.016,-24.299,21.445,-41.944
C09676=1018.102,82.053,-127.997,-24.298,21.444,-41.947
C09677=1018.105,81.842,-127.978,-24.298,21.445,-41.949
C09678=1018.107,81.630,-127.958,-24.298,21.445,-41.951
C09679=1018.109,81.417,-127.938,-24.297,21.445,-41.953
C09680=1018.111,81.204,-127.918,-24.297,21.445,-41.955
C09681=1018.113,80.992,-127.899,-24.297,21.445,-41.956
C09682=1018.115,80.779,-127.879,-24.297,21.446,-41.958
C09683=1018.117,80.566,-127.859,-24.296,21.446,-41.960
C09684=1018.119,80.354,-127.840,-24.296,21.446,-41.962
C09685=1018.121,80.142,-127.820,-24.296,21.446,-41.964
C09686=1018.122,79.932,-127.800,-24.296,21.447,-41.966
C09687=1018.127,79.518,-127.762,-24.295,21.447,-41.970
C09688=1018.131,79.112,-127.725,-24.294,21.447,-41.973
C09689=1018.134,78.715,-127.688,-24.294,21.447,-41.977
C09690=1018.138,78.324,-127.653,-24.293,21.448,-41.980
C09691=1018.141,77.938,-127.617,-24.293,21.447,-41.986
C09692=1018.145,77.551,-127.581,-24.292,21.448,-41.989
C09693=1018.148,77.163,-127.545,-24.292,21.449,-41.994
C09694=1018.152,76.768,-127.509,-24.291,21.449,-41.997
C09695=1018.155,76.366,-127.473,-24.291,21.449,-42.001
C09696=1018.159,75.955,-127.434,-24.290,21.450,-42.004
C09697=1018.162,75.535,-127.396,-24.290,21.450,-42.008
C09698=1018.164,75.322,-127.376,-24.289,21.451,-42.010
C09699=1018.166,75.109,-127.357,-24.289,21.451,-42.012
C09700=1018.168,74.895,-127.337,-24.289,21.450,-42.015
C09701=1018.170,74.682,-127.318,-24.288,21.451,-42.017
C09702=1018.172,74.468,-127.298,-24.288,21.451,-42.019
C09703=1018.174,74.256,-127.278,-24.288,21.451,-42.021
C09704=1018.176,74.044,-127.259,-24.288,21.451,-42.023
C09705=1018.177,73.832,-127.240,-24.287,21.452,-42.025
C09706=1018.181,73.412,-127.201,-24.287,21.452,-42.028
C09707=1018.185,72.995,-127.163,-24.286,21.452,-42.034
C09708=1018.188,72.578,-127.124,-24.285,21.452,-42.037
C09709=1018.191,72.165,-127.087,-24.285,21.453,-42.041
C09710=1018.195,71.753,-127.049,-24.285,21.453,-42.045
C09711=1018.199,71.342,-127.012,-24.284,21.454,-42.049
C09712=1018.203,70.931,-126.974,-24.283,21.453,-42.054
C09713=1018.206,70.520,-126.936,-24.283,21.454,-42.058
C09714=1018.209,70.109,-126.899,-24.282,21.454,-42.061
C09715=1018.212,69.698,-126.861,-24.282,21.455,-42.065
C09716=1018.216,69.288,-126.824,-24.281,21.455,-42.069
C09717=1018.219,68.878,-126.786,-24.280,21.455,-42.074
C09718=1018.222,68.471,-126.749,-24.280,21.456,-42.078
C09719=1018.226,68.065,-126.712,-24.279,21.456,-42.082
C09720=1018.229,67.661,-126.674,-24.279,21.457,-42.085
C09721=1018.232,67.258,-126.638,-24.278,21.457,-42.089
C09722=1018.235,66.855,-126.601,-24.278,21.457,-42.094
C09723=1018.239,66.454,-126.565,-24.277,21.457,-42.098
C09724=1018.241,66.056,-126.528,-24.277,21.458,-42.102
C09725=1018.245,65.648,-126.491,-24.276,21.458,-42.106
C09726=1018.247,65.436,-126.472,-24.276,21.459,-42.108
C09727=1018.249,65.214,-126.452,-24.275,21.458,-42.111
C09728=1018.250,64.984,-126.431,-24.275,21.458,-42.113
C09729=1018.252,64.748,-126.409,-24.275,21.459,-42.115
C09730=1018.254,64.512,-126.387,-24.274,21.459,-42.116
C09731=1018.256,64.283,-126.367,-24.274,21.459,-42.120
C09732=1018.258,64.065,-126.347,-24.274,21.460,-42.122
C09733=1018.259,63.858,-126.329,-24.274,21.460,-42.124
C09734=1018.261,63.641,-126.308,-24.273,21.459,-42.127
C09735=1018.263,63.391,-126.286,-24.273,21.460,-42.129
C09736=1018.265,63.123,-126.262,-24.272,21.460,-42.131
C09737=1018.266,62.870,-126.239,-24.272,21.460,-42.133
C09738=1018.270,62.450,-126.200,-24.271,21.461,-42.139
C09739=1018.273,62.050,-126.164,-24.271,21.461,-42.142
C09740=1018.276,61.650,-126.128,-24.270,21.462,-42.146
C09741=1018.278,61.250,-126.091,-24.270,21.462,-42.150
C09742=1018.282,60.850,-126.055,-24.269,21.462,-42.155
C09743=1018.285,60.450,-126.018,-24.269,21.463,-42.159
C09744=1018.288,60.049,-125.982,-24.268,21.463,-42.163
C09745=1018.291,59.649,-125.946,-24.268,21.464,-42.166
C09746=1018.293,59.249,-125.909,-24.267,21.463,-42.172
C09747=1018.296,58.849,-125.873,-24.266,21.464,-42.175
C09748=1018.299,58.449,-125.837,-24.266,21.464,-42.179
C09749=1018.302,58.049,-125.801,-24.265,21.465,-42.183
C09750=1018.305,57.648,-125.765,-24.264,21.465,-42.188
C09751=1018.308,57.247,-125.729,-24.264,21.465,-42.192
C09752=1018.311,56.848,-125.693,-24.264,21.466,-42.196
C09753=1018.314,56.448,-125.657,-24.263,21.465,-42.201
C09754=1018.316,56.047,-125.620,-24.262,21.467,-42.205
C09755=1018.319,55.647,-125.584,-24.262,21.467,-42.209
C09756=1018.322,55.247,-125.547,-24.261,21.468,-42.212
C09757=1018.325,54.847,-125.511,-24.260,21.468,-42.218
C09758=1018.327,54.447,-125.475,-24.260,21.468,-42.221
C09759=1018.330,54.046,-125.440,-24.259,21.468,-42.225
C09760=1018.333,53.646,-125.404,-24.259,21.468,-42.230
C09761=1018.336,53.246,-125.367,-24.258,21.469,-42.234
C09762=1018.339,52.846,-125.331,-24.258,21.469,-42.238
C09763=1018.340,52.446,-125.295,-24.257,21.469,-42.243
C09764=1018.343,52.046,-125.259,-24.256,21.470,-42.247
C09765=1018.346,51.645,-125.223,-24.256,21.471,-42.251
C09766=1018.348,51.216,-125.185,-24.255,21.471,-42.256
C09767=1018.351,50.845,-125.151,-24.255,21.471,-42.260
C09768=1018.354,50.445,-125.115,-24.254,21.472,-42.264
C09769=1018.356,50.045,-125.080,-24.254,21.472,-42.268
C09770=1018.359,49.645,-125.043,-24.253,21.472,-42.273
C09771=1018.361,49.245,-125.009,-24.252,21.473,-42.277
C09772=1018.364,48.844,-124.972,-24.251,21.472,-42.282
C09773=1018.366,48.444,-124.937,-24.251,21.474,-42.286
C09774=1018.369,48.044,-124.900,-24.251,21.474,-42.290
C09775=1018.371,47.644,-124.865,-24.250,21.474,-42.295
C09776=1018.374,47.245,-124.828,-24.249,21.475,-42.299
C09777=1018.376,46.844,-124.793,-24.249,21.475,-42.302
C09778=1018.379,46.444,-124.757,-24.248,21.475,-42.308
C09779=1018.381,46.044,-124.721,-24.247,21.475,-42.311
C09780=1018.383,45.644,-124.686,-24.247,21.477,-42.316
C09781=1018.386,45.243,-124.649,-24.246,21.477,-42.321
C09782=1018.388,44.843,-124.614,-24.246,21.477,-42.325
C09783=1018.390,44.443,-124.578,-24.245,21.477,-42.330
C09784=1018.393,44.043,-124.542,-24.244,21.477,-42.333
C09785=1018.396,43.644,-124.507,-24.244,21.479,-42.338
C09786=1018.397,43.243,-124.471,-24.243,21.479,-42.343
C09787=1018.400,42.843,-124.436,-24.243,21.479,-42.347
C09788=1018.402,42.443,-124.400,-24.242,21.479,-42.352
C09789=1018.405,42.043,-124.364,-24.241,21.479,-42.356
C09790=1018.407,41.644,-124.329,-24.241,21.480,-42.359
C09791=1018.409,41.243,-124.293,-24.240,21.481,-42.365
C09792=1018.411,40.843,-124.258,-24.240,21.481,-42.369
C09793=1018.413,40.443,-124.222,-24.239,21.481,-42.374
C09794=1018.415,40.043,-124.186,-24.238,21.481,-42.378
C09795=1018.418,39.644,-124.151,-24.238,21.482,-42.383
C09796=1018.419,39.244,-124.115,-24.237,21.483,-42.387
C09797=1018.422,38.844,-124.080,-24.237,21.483,-42.391
C09798=1018.424,38.444,-124.045,-24.236,21.483,-42.396
C09799=1018.426,38.044,-124.009,-24.235,21.483,-42.400
C09800=1018.428,37.645,-123.974,-24.235,21.484,-42.405
C09801=1018.430,37.245,-123.938,-24.234,21.485,-42.409
C09802=1018.432,36.844,-123.903,-24.233,21.484,-42.414
C09803=1018.434,36.445,-123.868,-24.233,21.485,-42.418
C09804=1018.437,36.045,-123.832,-24.232,21.486,-42.424
C09805=1018.438,35.645,-123.797,-24.231,21.486,-42.428
C09806=1018.440,35.246,-123.761,-24.231,21.486,-42.433
C09807=1018.443,34.845,-123.727,-24.230,21.486,-42.437
C09808=1018.444,34.446,-123.691,-24.229,21.487,-42.442
C09809=1018.446,34.046,-123.656,-24.229,21.488,-42.446
C09810=1018.448,33.646,-123.620,-24.228,21.487,-42.451
C09811=1018.450,33.247,-123.585,-24.228,21.489,-42.455
C09812=1018.452,32.847,-123.549,-24.227,21.489,-42.461
C09813=1018.454,32.447,-123.515,-24.226,21.489,-42.464
C09814=1018.456,32.048,-123.480,-24.226,21.489,-42.469
C09815=1018.457,31.648,-123.445,-24.225,21.490,-42.474
C09816=1018.459,31.248,-123.409,-24.224,21.490,-42.479
C09817=1018.461,30.849,-123.374,-24.224,21.491,-42.483
C09818=1018.462,30.450,-123.339,-24.223,21.491,-42.488
C09819=1018.465,30.050,-123.304,-24.223,21.492,-42.492
C09820=1018.467,29.650,-123.269,-24.222,21.492,-42.497
C09821=1018.468,29.251,-123.234,-24.221,21.492,-42.501
C09822=1018.470,28.851,-123.198,-24.221,21.493,-42.507
C09823=1018.471,28.452,-123.163,-24.220,21.493,-42.510
C09824=1018.473,28.052,-123.129,-24.219,21.493,-42.516
C09825=1018.475,27.653,-123.094,-24.219,21.495,-42.520
C09826=1018.477,27.253,-123.059,-24.218,21.494,-42.525
C09827=1018.479,26.854,-123.024,-24.218,21.495,-42.529
C09828=1018.480,26.455,-122.989,-24.217,21.496,-42.534
C09829=1018.482,26.055,-122.954,-24.216,21.496,-42.540
C09830=1018.484,25.656,-122.919,-24.215,21.496,-42.543
C09831=1018.485,25.257,-122.884,-24.215,21.497,-42.549
C09832=1018.487,24.858,-122.849,-24.214,21.497,-42.553
C09833=1018.488,24.459,-122.814,-24.213,21.497,-42.558
C09834=1018.489,24.075,-122.781,-24.213,21.498,-42.562
C09835=1018.491,23.745,-122.752,-24.213,21.498,-42.564
C09836=1018.492,23.473,-122.728,-24.212,21.498,-42.567
C09837=1018.492,23.238,-122.708,-24.211,21.499,-42.573
C09838=1018.493,23.007,-122.688,-24.211,21.500,-42.577
C09839=1018.495,22.740,-122.665,-24.211,21.500,-42.580
C09840=1018.495,22.419,-122.636,-24.210,21.500,-42.584
C09841=1018.498,22.044,-122.605,-24.210,21.501,-42.586
C09842=1018.499,21.630,-122.568,-24.209,21.501,-42.593
C09843=1018.499,21.386,-122.547,-24.208,21.501,-42.597
C09844=1018.501,21.114,-122.524,-24.208,21.502,-42.599
C09845=1018.502,20.822,-122.498,-24.207,21.501,-42.602
C09846=1018.503,20.525,-122.472,-24.207,21.501,-42.604
C09847=1018.503,20.237,-122.448,-24.207,21.503,-42.606
C09848=1018.504,19.973,-122.425,-24.206,21.502,-42.610
C09849=1018.505,19.736,-122.404,-24.206,21.503,-42.613
C09850=1018.506,19.525,-122.385,-24.205,21.503,-42.617
C09851=1018.508,19.127,-122.351,-24.205,21.503,-42.622
C09852=1018.508,18.731,-122.317,-24.204,21.503,-42.626
C09853=1018.510,18.336,-122.282,-24.203,21.504,-42.632
C09854=1018.512,17.941,-122.248,-24.203,21.505,-42.635
C09855=1018.513,17.546,-122.215,-24.202,21.505,-42.641
C09856=1018.514,17.153,-122.180,-24.201,21.505,-42.646
C09857=1018.515,16.760,-122.146,-24.201,21.506,-42.650
C09858=1018.517,16.368,-122.112,-24.200,21.506,-42.656
C09859=1018.518,15.977,-122.079,-24.200,21.507,-42.659
C09860=1018.519,15.587,-122.045,-24.199,21.507,-42.665
C09861=1018.520,15.198,-122.011,-24.198,21.508,-42.670
C09862=1018.521,14.809,-121.978,-24.198,21.508,-42.674
C09863=1018.523,14.421,-121.945,-24.197,21.509,-42.680
C09864=1018.523,14.032,-121.911,-24.196,21.509,-42.683
C09865=1018.525,13.646,-121.878,-24.196,21.509,-42.689
C09866=1018.526,13.259,-121.844,-24.195,21.511,-42.693
C09867=1018.526,12.872,-121.811,-24.194,21.510,-42.698
C09868=1018.528,12.485,-121.778,-24.193,21.510,-42.703
C09869=1018.528,12.099,-121.745,-24.193,21.512,-42.707
C09870=1018.530,11.713,-121.712,-24.192,21.511,-42.713
C09871=1018.531,11.328,-121.679,-24.192,21.512,-42.716
C09872=1018.531,10.944,-121.645,-24.191,21.513,-42.722
C09873=1018.533,10.563,-121.613,-24.191,21.513,-42.726
C09874=1018.533,10.185,-121.581,-24.190,21.513,-42.731
C09875=1018.535,9.808,-121.548,-24.189,21.514,-42.737
C09876=1018.535,9.433,-121.516,-24.189,21.514,-42.740
C09877=1018.536,9.056,-121.484,-24.188,21.515,-42.746
C09878=1018.537,8.678,-121.452,-24.187,21.515,-42.751
C09879=1018.538,8.298,-121.420,-24.187,21.516,-42.755
C09880=1018.539,7.913,-121.386,-24.186,21.516,-42.761
C09881=1018.539,7.526,-121.353,-24.185,21.517,-42.764
C09882=1018.541,7.136,-121.320,-24.185,21.517,-42.770
C09883=1018.541,6.743,-121.286,-24.184,21.517,-42.775
C09884=1018.542,6.350,-121.253,-24.183,21.519,-42.779
C09885=1018.543,5.956,-121.220,-24.182,21.518,-42.785
C09886=1018.543,5.562,-121.185,-24.182,21.519,-42.790
C09887=1018.544,5.167,-121.152,-24.181,21.520,-42.794
C09888=1018.546,4.771,-121.119,-24.180,21.519,-42.799
C09889=1018.546,4.375,-121.084,-24.180,21.520,-42.805
C09890=1018.547,3.987,-121.052,-24.179,21.521,-42.809
C09891=1018.548,3.627,-121.021,-24.179,21.521,-42.812
C09892=1018.548,3.299,-120.994,-24.178,21.521,-42.817
C09893=1018.548,2.985,-120.967,-24.177,21.522,-42.823
C09894=1018.549,2.663,-120.940,-24.177,21.522,-42.827
C09895=1018.550,2.310,-120.909,-24.176,21.523,-42.833
C09896=1018.550,1.924,-120.877,-24.175,21.524,-42.836
C09897=1018.552,1.526,-120.843,-24.175,21.523,-42.841
C09898=1018.552,1.128,-120.809,-24.174,21.525,-42.846
C09899=1018.552,0.727,-120.775,-24.173,21.525,-42.851
C09900=1018.553,0.326,-120.742,-24.173,21.525,-42.857
C09901=1018.553,-0.077,-120.708,-24.172,21.525,-42.862
C09902=1018.554,-0.483,-120.673,-24.171,21.526,-42.867
C09903=1018.554,-0.891,-120.638,-24.171,21.527,-42.872
C09904=1018.555,-1.301,-120.604,-24.170,21.527,-42.877
C09905=1018.556,-1.714,-120.569,-24.169,21.528,-42.882
C09906=1018.556,-2.129,-120.534,-24.169,21.529,-42.888
C09907=1018.557,-2.546,-120.500,-24.168,21.529,-42.893
C09908=1018.558,-2.965,-120.464,-24.167,21.529,-42.899
C09909=1018.558,-3.386,-120.429,-24.166,21.530,-42.904
C09910=1018.558,-3.598,-120.411,-24.166,21.530,-42.908
C09911=1018.558,-3.809,-120.393,-24.165,21.530,-42.910
C09912=1018.559,-4.024,-120.375,-24.165,21.530,-42.913
C09913=1018.559,-4.240,-120.357,-24.165,21.531,-42.915
C09914=1018.559,-4.456,-120.339,-24.164,21.531,-42.919
C09915=1018.559,-4.674,-120.321,-24.164,21.531,-42.921
C09916=1018.559,-4.895,-120.302,-24.163,21.532,-42.925
C09917=1018.560,-5.116,-120.284,-24.163,21.532,-42.927
C09918=1018.560,-5.338,-120.265,-24.163,21.532,-42.930
C09919=1018.560,-5.562,-120.246,-24.162,21.532,-42.934
C09920=1018.560,-5.786,-120.227,-24.162,21.533,-42.935
C09921=1018.560,-6.010,-120.208,-24.161,21.533,-42.939
C09922=1018.560,-6.234,-120.190,-24.161,21.533,-42.941
C09923=1018.560,-6.458,-120.171,-24.161,21.533,-42.944
C09924=1018.561,-6.682,-120.152,-24.160,21.534,-42.947
C09925=1018.561,-6.904,-120.133,-24.160,21.534,-42.950
C09926=1018.561,-7.126,-120.115,-24.160,21.535,-42.952
C09927=1018.561,-7.346,-120.097,-24.159,21.534,-42.956
C09928=1018.561,-7.564,-120.079,-24.159,21.535,-42.959
C09929=1018.561,-7.783,-120.060,-24.158,21.535,-42.961
C09930=1018.562,-8.000,-120.042,-24.158,21.536,-42.965
C09931=1018.562,-8.217,-120.024,-24.158,21.536,-42.967
C09932=1018.562,-8.434,-120.006,-24.157,21.536,-42.971
C09933=1018.562,-8.651,-119.988,-24.157,21.537,-42.973
C09934=1018.563,-8.867,-119.970,-24.156,21.536,-42.976
C09935=1018.562,-9.084,-119.952,-24.156,21.537,-42.980
C09936=1018.562,-9.300,-119.934,-24.156,21.537,-42.982
C09937=1018.562,-9.516,-119.915,-24.155,21.538,-42.985
C09938=1018.562,-9.732,-119.897,-24.155,21.538,-42.987
C09939=1018.562,-9.948,-119.880,-24.154,21.538,-42.991
C09940=1018.562,-10.164,-119.861,-24.154,21.539,-42.993
C09941=1018.563,-10.380,-119.843,-24.154,21.538,-42.996
C09942=1018.563,-10.594,-119.826,-24.153,21.539,-42.998
C09943=1018.563,-10.809,-119.808,-24.153,21.539,-43.002
C09944=1018.563,-11.022,-119.790,-24.152,21.539,-43.006
C09945=1018.563,-11.237,-119.772,-24.152,21.540,-43.007
C09946=1018.563,-11.450,-119.755,-24.152,21.540,-43.011
C09947=1018.563,-11.663,-119.737,-24.151,21.540,-43.013
C09948=1018.563,-11.875,-119.719,-24.151,21.540,-43.016
C09949=1018.563,-12.087,-119.702,-24.151,21.541,-43.019
C09950=1018.563,-12.299,-119.684,-24.150,21.541,-43.022
C09951=1018.563,-12.509,-119.667,-24.150,21.542,-43.024
C09952=1018.563,-12.929,-119.632,-24.149,21.542,-43.029
C09953=1018.564,-13.346,-119.597,-24.148,21.543,-43.035
C09954=1018.563,-13.761,-119.563,-24.148,21.543,-43.041
C09955=1018.563,-14.173,-119.529,-24.147,21.544,-43.046
C09956=1018.563,-14.581,-119.495,-24.146,21.544,-43.052
C09957=1018.563,-14.986,-119.461,-24.145,21.545,-43.057
C09958=1018.563,-15.389,-119.428,-24.145,21.545,-43.063
C09959=1018.563,-15.790,-119.395,-24.144,21.546,-43.068
C09960=1018.563,-16.190,-119.362,-24.143,21.546,-43.074
C09961=1018.563,-16.587,-119.329,-24.142,21.547,-43.079
C09962=1018.562,-16.986,-119.297,-24.142,21.548,-43.085
C09963=1018.562,-17.384,-119.264,-24.141,21.547,-43.090
C09964=1018.562,-17.794,-119.229,-24.140,21.548,-43.098
C09965=1018.562,-18.042,-119.209,-24.139,21.549,-43.101
C09966=1018.562,-18.331,-119.186,-24.139,21.549,-43.105
C09967=1018.561,-18.642,-119.160,-24.139,21.550,-43.107
C09968=1018.562,-18.953,-119.134,-24.139,21.550,-43.109
C09969=1018.561,-19.241,-119.110,-24.138,21.550,-43.113
C09970=1018.561,-19.491,-119.090,-24.138,21.551,-43.116
C09971=1018.561,-19.901,-119.056,-24.136,21.551,-43.123
C09972=1018.561,-20.299,-119.024,-24.136,21.552,-43.129
C09973=1018.561,-20.697,-118.991,-24.135,21.553,-43.135
C09974=1018.560,-21.094,-118.959,-24.134,21.552,-43.140
C09975=1018.560,-21.491,-118.926,-24.134,21.553,-43.146
C09976=1018.560,-21.889,-118.893,-24.133,21.554,-43.151
C09977=1018.559,-22.286,-118.861,-24.132,21.554,-43.156
C09978=1018.559,-22.684,-118.828,-24.131,21.555,-43.162
C09979=1018.558,-23.081,-118.796,-24.131,21.555,-43.168
C09980=1018.558,-23.479,-118.763,-24.130,21.556,-43.173
C09981=1018.557,-23.876,-118.731,-24.129,21.556,-43.178
C09982=1018.557,-24.274,-118.698,-24.128,21.557,-43.184
C09983=1018.556,-24.672,-118.666,-24.128,21.558,-43.190
C09984=1018.555,-25.069,-118.634,-24.127,21.558,-43.195
C09985=1018.555,-25.467,-118.601,-24.126,21.558,-43.201
C09986=1018.555,-25.864,-118.569,-24.125,21.559,-43.206
C09987=1018.554,-26.261,-118.537,-24.125,21.560,-43.212
C09988=1018.554,-26.659,-118.504,-24.124,21.560,-43.217
C09989=1018.553,-27.056,-118.472,-24.123,21.561,-43.221
C09990=1018.552,-27.453,-118.440,-24.123,21.562,-43.227
C09991=1018.551,-27.851,-118.407,-24.122,21.562,-43.232
C09992=1018.551,-28.249,-118.375,-24.121,21.562,-43.238
C09993=1018.550,-28.647,-118.343,-24.120,21.563,-43.243
C09994=1018.550,-29.044,-118.311,-24.120,21.564,-43.249
C09995=1018.549,-29.441,-118.279,-24.119,21.565,-43.255
C09996=1018.548,-29.838,-118.247,-24.118,21.565,-43.260
//INST
///DATE 2021/06/17 16:00
///ATTR SC,RW,RJ
////FRAME ROBOT
///GROUP1 RB1
NOP
MOVL C00000 V=800.0 PL=0
MOVL C00001 V=800.0 PL=0
MOVL C00002 V=800.0 PL=0
MOVL C00003 V=800.0 PL=0
MOVL C00004 V=800.0 PL=0
MOVL C00005 V=800.0 PL=0
MOVL C00006 V=800.0 PL=0
MOVL C00007 V=800.0 PL=0
MOVL C00008 V=800.0 PL=0
MOVL C00009 V=800.0 PL=0
MOVL C00010 V=800.0 PL=0
MOVL C00011 V=800.0 PL=0
MOVL C00012 V=800.0 PL=0
MOVL C00013 V=800.0 PL=0
MOVL C00014 V=800.0 PL=0
MOVL C00015 V=800.0 PL=0
MOVL C00016 V=800.0 PL=0
MOVL C00017 V=800.0 PL=0
MOVL C00018 V=800.0 PL=0
MOVL C00019 V=800.0 PL=0
MOVL C00020 V=800.0 PL=0
MOVL C00021 V=800.0 PL=0
MOVL C00022 V=800.0 PL=0
MOVL C00023 V=800.0 PL=0
MOVL C00024 V=800.0 PL=0
MOVL C00025 V=800.0 PL=0
MOVL C00026 V=800.0 PL=0
MOVL C00027 V=800.0 PL=0
MOVL C00028 V=800.0 PL=0
MOVL C00029 V=800.0 PL=0
MOVL C00030 V=800.0 PL=0
MOVL C00031 V=800.0 PL=0
MOVL C00032 V=800.0 PL=0
MOVL C00033 V=800.0 PL=0
MOVL C00034 V=800.0 PL=0
MOVL C00035 V=800.0 PL=0
MOVL C00036 V=800.0 PL=0
MOVL C00037 V=800.0 PL=0
MOVL C00038 V=800.0 PL=0
MOVL C00039 V=800.0 PL=0
MOVL C00040 V=800.0 PL=0
MOVL C00041 V=800.0 PL=0
MOVL C00042 V=800.0 PL=0
MOVL C00043 V=800.0 PL=0
MOVL C00044 V=800.0 PL=0
MOVL C00045 V=800.0 PL=0
MOVL C00046 V=800.0 PL=0
MOVL C00047 V=800.0 PL=0
MOVL C00048 V=800.0 PL=0
MOVL C00049 V=800.0 PL=0
MOVL C00050 V=800.0 PL=0
MOVL C00051 V=800.0 PL=0
MOVL C00052 V=800.0 PL=0
MOVL C00053 V=800.0 PL=0
MOVL C00054 V=800.0 PL=0
MOVL C00055 V=800.0 PL=0
MOVL C00056 V=800.0 PL=0
MOVL C00057 V=800.0 PL=0
MOVL C00058 V=800.0 PL=0
MOVL C00059 V=800.0 PL=0
MOVL C00060 V=800.0 PL=0
MOVL C00061 V=800.0 PL=0
MOVL C00062 V=800.0 PL=0
MOVL C00063 V=800.0 PL=0
MOVL C00064 V=800.0 PL=0
MOVL C00065 V=800.0 PL=0
MOVL C00066 V=800.0 PL=0
MOVL C00067 V=800.0 PL=0
MOVL C00068 V=800.0 PL=0
MOVL C00069 V=800.0 PL=0
MOVL C00070 V=800.0 PL=0
MOVL C00071 V=800.0 PL=0
MOVL C00072 V=800.0 PL=0
MOVL C00073 V=800.0 PL=0
MOVL C00074 V=800.0 PL=0
MOVL C00075 V=800.0 PL=0
MOVL C00076 V=800.0 PL=0
MOVL C00077 V=800.0 PL=0
MOVL C00078 V=800.0 PL=0
MOVL C00079 V=800.0 PL=0
MOVL C00080 V=800.0 PL=0
MOVL C00081 V=800.0 PL=0
MOVL C00082 V=800.0 PL=0
MOVL C00083 V=800.0 PL=0
MOVL C00084 V=800.0 PL=0
MOVL C00085 V=800.0 PL=0
MOVL C00086 V=800.0 PL=0
MOVL C00087 V=800.0 PL=0
MOVL C00088 V=800.0 PL=0
MOVL C00089 V=800.0 PL=0
MOVL C00090 V=800.0 PL=0
MOVL C00091 V=800.0 PL=0
MOVL C00092 V=800.0 PL=0
MOVL C00093 V=800.0 PL=0
MOVL C00094 V=800.0 PL=0
MOVL C00095 V=800.0 PL=0
MOVL C00096 V=800.0 PL=0
MOVL C00097 V=800.0 PL=0
MOVL C00098 V=800.0 PL=0
MOVL C00099 V=800.0 PL=0
MOVL C00100 V=800.0 PL=0
MOVL C00101 V=800.0 PL=0
MOVL C00102 V=800.0 PL=0
MOVL C00103 V=800.0 PL=0
MOVL C00104 V=800.0 PL=0
MOVL C00105 V=800.0 PL=0
MOVL C00106 V=800.0 PL=0
MOVL C00107 V=800.0 PL=0
MOVL C00108 V=800.0 PL=0
MOVL C00109 V=800.0 PL=0
MOVL C00110 V=800.0 PL=0
MOVL C00111 V=800.0 PL=0
MOVL C00112 V=800.0 PL=0
MOVL C00113 V=800.0 PL=0
MOVL C00114 V=800.0 PL=0
MOVL C00115 V=800.0 PL=0
MOVL C00116 V=800.0 PL=0
MOVL C00117 V=800.0 PL=0
MOVL C00118 V=800.0 PL=0
MOVL C00119 V=800.0 PL=0
MOVL C00120 V=800.0 PL=0
MOVL C00121 V=800.0 PL=0
MOVL C00122 V=800.0 PL=0
MOVL C00123 V=800.0 PL=0
MOVL C00124 V=800.0 PL=0
MOVL C00125 V=800.0 PL=0
MOVL C00126 V=800.0 PL=0
MOVL C00127 V=800.0 PL=0
MOVL C00128 V=800.0 PL=0
MOVL C00129 V=800.0 PL=0
MOVL C00130 V=800.0 PL=0
MOVL C00131 V=800.0 PL=0
MOVL C00132 V=800.0 PL=0
MOVL C00133 V=800.0 PL=0
MOVL C00134 V=800.0 PL=0
MOVL C00135 V=800.0 PL=0
MOVL C00136 V=800.0 PL=0
MOVL C00137 V=800.0 PL=0
MOVL C00138 V=800.0 PL=0
MOVL C00139 V=800.0 PL=0
MOVL C00140 V=800.0 PL=0
MOVL C00141 V=800.0 PL=0
MOVL C00142 V=800.0 PL=0
MOVL C00143 V=800.0 PL=0
MOVL C00144 V=800.0 PL=0
MOVL C00145 V=800.0 PL=0
MOVL C00146 V=800.0 PL=0
MOVL C00147 V=800.0 PL=0
MOVL C00148 V=800.0 PL=0
MOVL C00149 V=800.0 PL=0
MOVL C00150 V=800.0 PL=0
MOVL C00151 V=800.0 PL=0
MOVL C00152 V=800.0 PL=0
MOVL C00153 V=800.0 PL=0
MOVL C00154 V=800.0 PL=0
MOVL C00155 V=800.0 PL=0
MOVL C00156 V=800.0 PL=0
MOVL C00157 V=800.0 PL=0
MOVL C00158 V=800.0 PL=0
MOVL C00159 V=800.0 PL=0
MOVL C00160 V=800.0 PL=0
MOVL C00161 V=800.0 PL=0
MOVL C00162 V=800.0 PL=0
MOVL C00163 V=800.0 PL=0
MOVL C00164 V=800.0 PL=0
MOVL C00165 V=800.0 PL=0
MOVL C00166 V=800.0 PL=0
MOVL C00167 V=800.0 PL=0
MOVL C00168 V=800.0 PL=0
MOVL C00169 V=800.0 PL=0
MOVL C00170 V=800.0 PL=0
MOVL C00171 V=800.0 PL=0
MOVL C00172 V=800.0 PL=0
MOVL C00173 V=800.0 PL=0
MOVL C00174 V=800.0 PL=0
MOVL C00175 V=800.0 PL=0
MOVL C00176 V=800.0 PL=0
MOVL C00177 V=800.0 PL=0
MOVL C00178 V=800.0 PL=0
MOVL C00179 V=800.0 PL=0
MOVL C00180 V=800.0 PL=0
MOVL C00181 V=800.0 PL=0
MOVL C00182 V=800.0 PL=0
MOVL C00183 V=800.0 PL=0
MOVL C00184 V=800.0 PL=0
MOVL C00185 V=800.0 PL=0
MOVL C00186 V=800.0 PL=0
MOVL C00187 V=800.0 PL=0
MOVL C00188 V=800.0 PL=0
MOVL C00189 V=800.0 PL=0
MOVL C00190 V=800.0 PL=0
MOVL C00191 V=800.0 PL=0
MOVL C00192 V=800.0 PL=0
MOVL C00193 V=800.0 PL=0
MOVL C00194 V=800.0 PL=0
MOVL C00195 V=800.0 PL=0
MOVL C00196 V=800.0 PL=0
MOVL C00197 V=800.0 PL=0
MOVL C00198 V=800.0 PL=0
MOVL C00199 V=800.0 PL=0
MOVL C00200 V=800.0 PL=0
MOVL C00201 V=800.0 PL=0
MOVL C00202 V=800.0 PL=0
MOVL C00203 V=800.0 PL=0
MOVL C00204 V=800.0 PL=0
MOVL C00205 V=800.0 PL=0
MOVL C00206 V=800.0 PL=0
MOVL C00207 V=800.0 PL=0
MOVL C00208 V=800.0 PL=0
MOVL C00209 V=800.0 PL=0
MOVL C00210 V=800.0 PL=0
MOVL C00211 V=800.0 PL=0
MOVL C00212 V=800.0 PL=0
MOVL C00213 V=800.0 PL=0
MOVL C00214 V=800.0 PL=0
MOVL C00215 V=800.0 PL=0
MOVL C00216 V=800.0 PL=0
MOVL C00217 V=800.0 PL=0
MOVL C00218 V=800.0 PL=0
MOVL C00219 V=800.0 PL=0
MOVL C00220 V=800.0 PL=0
MOVL C00221 V=800.0 PL=0
MOVL C00222 V=800.0 PL=0
MOVL C00223 V=800.0 PL=0
MOVL C00224 V=800.0 PL=0
MOVL C00225 V=800.0 PL=0
MOVL C00226 V=800.0 PL=0
MOVL C00227 V=800.0 PL=0
MOVL C00228 V=800.0 PL=0
MOVL C00229 V=800.0 PL=0
MOVL C00230 V=800.0 PL=0
MOVL C00231 V=800.0 PL=0
MOVL C00232 V=800.0 PL=0
MOVL C00233 V=800.0 PL=0
MOVL C00234 V=800.0 PL=0
MOVL C00235 V=800.0 PL=0
MOVL C00236 V=800.0 PL=0
MOVL C00237 V=800.0 PL=0
MOVL C00238 V=800.0 PL=0
MOVL C00239 V=800.0 PL=0
MOVL C00240 V=800.0 PL=0
MOVL C00241 V=800.0 PL=0
MOVL C00242 V=800.0 PL=0
MOVL C00243 V=800.0 PL=0
MOVL C00244 V=800.0 PL=0
MOVL C00245 V=800.0 PL=0
MOVL C00246 V=800.0 PL=0
MOVL C00247 V=800.0 PL=0
MOVL C00248 V=800.0 PL=0
MOVL C00249 V=800.0 PL=0
MOVL C00250 V=800.0 PL=0
MOVL C00251 V=800.0 PL=0
MOVL C00252 V=800.0 PL=0
MOVL C00253 V=800.0 PL=0
MOVL C00254 V=800.0 PL=0
MOVL C00255 V=800.0 PL=0
MOVL C00256 V=800.0 PL=0
MOVL C00257 V=800.0 PL=0
MOVL C00258 V=800.0 PL=0
MOVL C00259 V=800.0 PL=0
MOVL C00260 V=800.0 PL=0
MOVL C00261 V=800.0 PL=0
MOVL C00262 V=800.0 PL=0
MOVL C00263 V=800.0 PL=0
MOVL C00264 V=800.0 PL=0
MOVL C00265 V=800.0 PL=0
MOVL C00266 V=800.0 PL=0
MOVL C00267 V=800.0 PL=0
MOVL C00268 V=800.0 PL=0
MOVL C00269 V=800.0 PL=0
MOVL C00270 V=800.0 PL=0
MOVL C00271 V=800.0 PL=0
MOVL C00272 V=800.0 PL=0
MOVL C00273 V=800.0 PL=0
MOVL C00274 V=800.0 PL=0
MOVL C00275 V=800.0 PL=0
MOVL C00276 V=800.0 PL=0
MOVL C00277 V=800.0 PL=0
MOVL C00278 V=800.0 PL=0
MOVL C00279 V=800.0 PL=0
MOVL C00280 V=800.0 PL=0
MOVL C00281 V=800.0 PL=0
MOVL C00282 V=800.0 PL=0
MOVL C00283 V=800.0 PL=0
MOVL C00284 V=800.0 PL=0
MOVL C00285 V=800.0 PL=0
MOVL C00286 V=800.0 PL=0
MOVL C00287 V=800.0 PL=0
MOVL C00288 V=800.0 PL=0
MOVL C00289 V=800.0 PL=0
MOVL C00290 V=800.0 PL=0
MOVL C00291 V=800.0 PL=0
MOVL C00292 V=800.0 PL=0
MOVL C00293 V=800.0 PL=0
MOVL C00294 V=800.0 PL=0
MOVL C00295 V=800.0 PL=0
MOVL C00296 V=800.0 PL=0
MOVL C00297 V=800.0 PL=0
MOVL C00298 V=800.0 PL=0
MOVL C00299 V=800.0 PL=0
MOVL C00300 V=800.0 PL=0
MOVL C00301 V=800.0 PL=0
MOVL C00302 V=800.0 PL=0
MOVL C00303 V=800.0 PL=0
MOVL C00304 V=800.0 PL=0
MOVL C00305 V=800.0 PL=0
MOVL C00306 V=800.0 PL=0
MOVL C00307 V=800.0 PL=0
MOVL C00308 V=800.0 PL=0
MOVL C00309 V=800.0 PL=0
MOVL C00310 V=800.0 PL=0
MOVL C00311 V=800.0 PL=0
MOVL C00312 V=800.0 PL=0
MOVL C00313 V=800.0 PL=0
MOVL C00314 V=800.0 PL=0
MOVL C00315 V=800.0 PL=0
MOVL C00316 V=800.0 PL=0
MOVL C00317 V=800.0 PL=0
MOVL C00318 V=800.0 PL=0
MOVL C00319 V=800.0 PL=0
MOVL C00320 V=800.0 PL=0
MOVL C00321 V=800.0 PL=0
MOVL C00322 V=800.0 PL=0
MOVL C00323 V=800.0 PL=0
MOVL C00324 V=800.0 PL=0
MOVL C00325 V=800.0 PL=0
MOVL C00326 V=800.0 PL=0
MOVL C00327 V=800.0 PL=0
MOVL C00328 V=800.0 PL=0
MOVL C00329 V=800.0 PL=0
MOVL C00330 V=800.0 PL=0
MOVL C00331 V=800.0 PL=0
MOVL C00332 V=800.0 PL=0
MOVL C00333 V=800.0 PL=0
MOVL C00334 V=800.0 PL=0
MOVL C00335 V=800.0 PL=0
MOVL C00336 V=800.0 PL=0
MOVL C00337 V=800.0 PL=0
MOVL C00338 V=800.0 PL=0
MOVL C00339 V=800.0 PL=0
MOVL C00340 V=800.0 PL=0
MOVL C00341 V=800.0 PL=0
MOVL C00342 V=800.0 PL=0
MOVL C00343 V=800.0 PL=0
MOVL C00344 V=800.0 PL=0
MOVL C00345 V=800.0 PL=0
MOVL C00346 V=800.0 PL=0
MOVL C00347 V=800.0 PL=0
MOVL C00348 V=800.0 PL=0
MOVL C00349 V=800.0 PL=0
MOVL C00350 V=800.0 PL=0
MOVL C00351 V=800.0 PL=0
MOVL C00352 V=800.0 PL=0
MOVL C00353 V=800.0 PL=0
MOVL C00354 V=800.0 PL=0
MOVL C00355 V=800.0 PL=0
MOVL C00356 V=800.0 PL=0
MOVL C00357 V=800.0 PL=0
MOVL C00358 V=800.0 PL=0
MOVL C00359 V=800.0 PL=0
MOVL C00360 V=800.0 PL=0
MOVL C00361 V=800.0 PL=0
MOVL C00362 V=800.0 PL=0
MOVL C00363 V=800.0 PL=0
MOVL C00364 V=800.0 PL=0
MOVL C00365 V=800.0 PL=0
MOVL C00366 V=800.0 PL=0
MOVL C00367 V=800.0 PL=0
MOVL C00368 V=800.0 PL=0
MOVL C00369 V=800.0 PL=0
MOVL C00370 V=800.0 PL=0
MOVL C00371 V=800.0 PL=0
MOVL C00372 V=800.0 PL=0
MOVL C00373 V=800.0 PL=0
MOVL C00374 V=800.0 PL=0
MOVL C00375 V=800.0 PL=0
MOVL C00376 V=800.0 PL=0
MOVL C00377 V=800.0 PL=0
MOVL C00378 V=800.0 PL=0
MOVL C00379 V=800.0 PL=0
MOVL C00380 V=800.0 PL=0
MOVL C00381 V=800.0 PL=0
MOVL C00382 V=800.0 PL=0
MOVL C00383 V=800.0 PL=0
MOVL C00384 V=800.0 PL=0
MOVL C00385 V=800.0 PL=0
MOVL C00386 V=800.0 PL=0
MOVL C00387 V=800.0 PL=0
MOVL C00388 V=800.0 PL=0
MOVL C00389 V=800.0 PL=0
MOVL C00390 V=800.0 PL=0
MOVL C00391 V=800.0 PL=0
MOVL C00392 V=800.0 PL=0
MOVL C00393 V=800.0 PL=0
MOVL C00394 V=800.0 PL=0
MOVL C00395 V=800.0 PL=0
MOVL C00396 V=800.0 PL=0
MOVL C00397 V=800.0 PL=0
MOVL C00398 V=800.0 PL=0
MOVL C00399 V=800.0 PL=0
MOVL C00400 V=800.0 PL=0
MOVL C00401 V=800.0 PL=0
MOVL C00402 V=800.0 PL=0
MOVL C00403 V=800.0 PL=0
MOVL C00404 V=800.0 PL=0
MOVL C00405 V=800.0 PL=0
MOVL C00406 V=800.0 PL=0
MOVL C00407 V=800.0 PL=0
MOVL C00408 V=800.0 PL=0
MOVL C00409 V=800.0 PL=0
MOVL C00410 V=800.0 PL=0
MOVL C00411 V=800.0 PL=0
MOVL C00412 V=800.0 PL=0
MOVL C00413 V=800.0 PL=0
MOVL C00414 V=800.0 PL=0
MOVL C00415 V=800.0 PL=0
MOVL C00416 V=800.0 PL=0
MOVL C00417 V=800.0 PL=0
MOVL C00418 V=800.0 PL=0
MOVL C00419 V=800.0 PL=0
MOVL C00420 V=800.0 PL=0
MOVL C00421 V=800.0 PL=0
MOVL C00422 V=800.0 PL=0
MOVL C00423 V=800.0 PL=0
MOVL C00424 V=800.0 PL=0
MOVL C00425 V=800.0 PL=0
MOVL C00426 V=800.0 PL=0
MOVL C00427 V=800.0 PL=0
MOVL C00428 V=800.0 PL=0
MOVL C00429 V=800.0 PL=0
MOVL C00430 V=800.0 PL=0
MOVL C00431 V=800.0 PL=0
MOVL C00432 V=800.0 PL=0
MOVL C00433 V=800.0 PL=0
MOVL C00434 V=800.0 PL=0
MOVL C00435 V=800.0 PL=0
MOVL C00436 V=800.0 PL=0
MOVL C00437 V=800.0 PL=0
MOVL C00438 V=800.0 PL=0
MOVL C00439 V=800.0 PL=0
MOVL C00440 V=800.0 PL=0
MOVL C00441 V=800.0 PL=0
MOVL C00442 V=800.0 PL=0
MOVL C00443 V=800.0 PL=0
MOVL C00444 V=800.0 PL=0
MOVL C00445 V=800.0 PL=0
MOVL C00446 V=800.0 PL=0
MOVL C00447 V=800.0 PL=0
MOVL C00448 V=800.0 PL=0
MOVL C00449 V=800.0 PL=0
MOVL C00450 V=800.0 PL=0
MOVL C00451 V=800.0 PL=0
MOVL C00452 V=800.0 PL=0
MOVL C00453 V=800.0 PL=0
MOVL C00454 V=800.0 PL=0
MOVL C00455 V=800.0 PL=0
MOVL C00456 V=800.0 PL=0
MOVL C00457 V=800.0 PL=0
MOVL C00458 V=800.0 PL=0
MOVL C00459 V=800.0 PL=0
MOVL C00460 V=800.0 PL=0
MOVL C00461 V=800.0 PL=0
MOVL C00462 V=800.0 PL=0
MOVL C00463 V=800.0 PL=0
MOVL C00464 V=800.0 PL=0
MOVL C00465 V=800.0 PL=0
MOVL C00466 V=800.0 PL=0
MOVL C00467 V=800.0 PL=0
MOVL C00468 V=800.0 PL=0
MOVL C00469 V=800.0 PL=0
MOVL C00470 V=800.0 PL=0
MOVL C00471 V=800.0 PL=0
MOVL C00472 V=800.0 PL=0
MOVL C00473 V=800.0 PL=0
MOVL C00474 V=800.0 PL=0
MOVL C00475 V=800.0 PL=0
MOVL C00476 V=800.0 PL=0
MOVL C00477 V=800.0 PL=0
MOVL C00478 V=800.0 PL=0
MOVL C00479 V=800.0 PL=0
MOVL C00480 V=800.0 PL=0
MOVL C00481 V=800.0 PL=0
MOVL C00482 V=800.0 PL=0
MOVL C00483 V=800.0 PL=0
MOVL C00484 V=800.0 PL=0
MOVL C00485 V=800.0 PL=0
MOVL C00486 V=800.0 PL=0
MOVL C00487 V=800.0 PL=0
MOVL C00488 V=800.0 PL=0
MOVL C00489 V=800.0 PL=0
MOVL C00490 V=800.0 PL=0
MOVL C00491 V=800.0 PL=0
MOVL C00492 V=800.0 PL=0
MOVL C00493 V=800.0 PL=0
MOVL C00494 V=800.0 PL=0
MOVL C00495 V=800.0 PL=0
MOVL C00496 V=800.0 PL=0
MOVL C00497 V=800.0 PL=0
MOVL C00498 V=800.0 PL=0
MOVL C00499 V=800.0 PL=0
MOVL C00500 V=800.0 PL=0
MOVL C00501 V=800.0 PL=0
MOVL C00502 V=800.0 PL=0
MOVL C00503 V=800.0 PL=0
MOVL C00504 V=800.0 PL=0
MOVL C00505 V=800.0 PL=0
MOVL C00506 V=800.0 PL=0
MOVL C00507 V=800.0 PL=0
MOVL C00508 V=800.0 PL=0
MOVL C00509 V=800.0 PL=0
MOVL C00510 V=800.0 PL=0
MOVL C00511 V=800.0 PL=0
MOVL C00512 V=800.0 PL=0
MOVL C00513 V=800.0 PL=0
MOVL C00514 V=800.0 PL=0
MOVL C00515 V=800.0 PL=0
MOVL C00516 V=800.0 PL=0
MOVL C00517 V=800.0 PL=0
MOVL C00518 V=800.0 PL=0
MOVL C00519 V=800.0 PL=0
MOVL C00520 V=800.0 PL=0
MOVL C00521 V=800.0 PL=0
MOVL C00522 V=800.0 PL=0
MOVL C00523 V=800.0 PL=0
MOVL C00524 V=800.0 PL=0
MOVL C00525 V=800.0 PL=0
MOVL C00526 V=800.0 PL=0
MOVL C00527 V=800.0 PL=0
MOVL C00528 V=800.0 PL=0
MOVL C00529 V=800.0 PL=0
MOVL C00530 V=800.0 PL=0
MOVL C00531 V=800.0 PL=0
MOVL C00532 V=800.0 PL=0
MOVL C00533 V=800.0 PL=0
MOVL C00534 V=800.0 PL=0
MOVL C00535 V=800.0 PL=0
MOVL C00536 V=800.0 PL=0
MOVL C00537 V=800.0 PL=0
MOVL C00538 V=800.0 PL=0
MOVL C00539 V=800.0 PL=0
MOVL C00540 V=800.0 PL=0
MOVL C00541 V=800.0 PL=0
MOVL C00542 V=800.0 PL=0
MOVL C00543 V=800.0 PL=0
MOVL C00544 V=800.0 PL=0
MOVL C00545 V=800.0 PL=0
MOVL C00546 V=800.0 PL=0
MOVL C00547 V=800.0 PL=0
MOVL C00548 V=800.0 PL=0
MOVL C00549 V=800.0 PL=0
MOVL C00550 V=800.0 PL=0
MOVL C00551 V=800.0 PL=0
MOVL C00552 V=800.0 PL=0
MOVL C00553 V=800.0 PL=0
MOVL C00554 V=800.0 PL=0
MOVL C00555 V=800.0 PL=0
MOVL C00556 V=800.0 PL=0
MOVL C00557 V=800.0 PL=0
MOVL C00558 V=800.0 PL=0
MOVL C00559 V=800.0 PL=0
MOVL C00560 V=800.0 PL=0
MOVL C00561 V=800.0 PL=0
MOVL C00562 V=800.0 PL=0
MOVL C00563 V=800.0 PL=0
MOVL C00564 V=800.0 PL=0
MOVL C00565 V=800.0 PL=0
MOVL C00566 V=800.0 PL=0
MOVL C00567 V=800.0 PL=0
MOVL C00568 V=800.0 PL=0
MOVL C00569 V=800.0 PL=0
MOVL C00570 V=800.0 PL=0
MOVL C00571 V=800.0 PL=0
MOVL C00572 V=800.0 PL=0
MOVL C00573 V=800.0 PL=0
MOVL C00574 V=800.0 PL=0
MOVL C00575 V=800.0 PL=0
MOVL C00576 V=800.0 PL=0
MOVL C00577 V=800.0 PL=0
MOVL C00578 V=800.0 PL=0
MOVL C00579 V=800.0 PL=0
MOVL C00580 V=800.0 PL=0
MOVL C00581 V=800.0 PL=0
MOVL C00582 V=800.0 PL=0
MOVL C00583 V=800.0 PL=0
MOVL C00584 V=800.0 PL=0
MOVL C00585 V=800.0 PL=0
MOVL C00586 V=800.0 PL=0
MOVL C00587 V=800.0 PL=0
MOVL C00588 V=800.0 PL=0
MOVL C00589 V=800.0 PL=0
MOVL C00590 V=800.0 PL=0
MOVL C00591 V=800.0 PL=0
MOVL C00592 V=800.0 PL=0
MOVL C00593 V=800.0 PL=0
MOVL C00594 V=800.0 PL=0
MOVL C00595 V=800.0 PL=0
MOVL C00596 V=800.0 PL=0
MOVL C00597 V=800.0 PL=0
MOVL C00598 V=800.0 PL=0
MOVL C00599 V=800.0 PL=0
MOVL C00600 V=800.0 PL=0
MOVL C00601 V=800.0 PL=0
MOVL C00602 V=800.0 PL=0
MOVL C00603 V=800.0 PL=0
MOVL C00604 V=800.0 PL=0
MOVL C00605 V=800.0 PL=0
MOVL C00606 V=800.0 PL=0
MOVL C00607 V=800.0 PL=0
MOVL C00608 V=800.0 PL=0
MOVL C00609 V=800.0 PL=0
MOVL C00610 V=800.0 PL=0
MOVL C00611 V=800.0 PL=0
MOVL C00612 V=800.0 PL=0
MOVL C00613 V=800.0 PL=0
MOVL C00614 V=800.0 PL=0
MOVL C00615 V=800.0 PL=0
MOVL C00616 V=800.0 PL=0
MOVL C00617 V=800.0 PL=0
MOVL C00618 V=800.0 PL=0
MOVL C00619 V=800.0 PL=0
MOVL C00620 V=800.0 PL=0
MOVL C00621 V=800.0 PL=0
MOVL C00622 V=800.0 PL=0
MOVL C00623 V=800.0 PL=0
MOVL C00624 V=800.0 PL=0
MOVL C00625 V=800.0 PL=0
MOVL C00626 V=800.0 PL=0
MOVL C00627 V=800.0 PL=0
MOVL C00628 V=800.0 PL=0
MOVL C00629 V=800.0 PL=0
MOVL C00630 V=800.0 PL=0
MOVL C00631 V=800.0 PL=0
MOVL C00632 V=800.0 PL=0
MOVL C00633 V=800.0 PL=0
MOVL C00634 V=800.0 PL=0
MOVL C00635 V=800.0 PL=0
MOVL C00636 V=800.0 PL=0
MOVL C00637 V=800.0 PL=0
MOVL C00638 V=800.0 PL=0
MOVL C00639 V=800.0 PL=0
MOVL C00640 V=800.0 PL=0
MOVL C00641 V=800.0 PL=0
MOVL C00642 V=800.0 PL=0
MOVL C00643 V=800.0 PL=0
MOVL C00644 V=800.0 PL=0
MOVL C00645 V=800.0 PL=0
MOVL C00646 V=800.0 PL=0
MOVL C00647 V=800.0 PL=0
MOVL C00648 V=800.0 PL=0
MOVL C00649 V=800.0 PL=0
MOVL C00650 V=800.0 PL=0
MOVL C00651 V=800.0 PL=0
MOVL C00652 V=800.0 PL=0
MOVL C00653 V=800.0 PL=0
MOVL C00654 V=800.0 PL=0
MOVL C00655 V=800.0 PL=0
MOVL C00656 V=800.0 PL=0
MOVL C00657 V=800.0 PL=0
MOVL C00658 V=800.0 PL=0
MOVL C00659 V=800.0 PL=0
MOVL C00660 V=800.0 PL=0
MOVL C00661 V=800.0 PL=0
MOVL C00662 V=800.0 PL=0
MOVL C00663 V=800.0 PL=0
MOVL C00664 V=800.0 PL=0
MOVL C00665 V=800.0 PL=0
MOVL C00666 V=800.0 PL=0
MOVL C00667 V=800.0 PL=0
MOVL C00668 V=800.0 PL=0
MOVL C00669 V=800.0 PL=0
MOVL C00670 V=800.0 PL=0
MOVL C00671 V=800.0 PL=0
MOVL C00672 V=800.0 PL=0
MOVL C00673 V=800.0 PL=0
MOVL C00674 V=800.0 PL=0
MOVL C00675 V=800.0 PL=0
MOVL C00676 V=800.0 PL=0
MOVL C00677 V=800.0 PL=0
MOVL C00678 V=800.0 PL=0
MOVL C00679 V=800.0 PL=0
MOVL C00680 V=800.0 PL=0
MOVL C00681 V=800.0 PL=0
MOVL C00682 V=800.0 PL=0
MOVL C00683 V=800.0 PL=0
MOVL C00684 V=800.0 PL=0
MOVL C00685 V=800.0 PL=0
MOVL C00686 V=800.0 PL=0
MOVL C00687 V=800.0 PL=0
MOVL C00688 V=800.0 PL=0
MOVL C00689 V=800.0 PL=0
MOVL C00690 V=800.0 PL=0
MOVL C00691 V=800.0 PL=0
MOVL C00692 V=800.0 PL=0
MOVL C00693 V=800.0 PL=0
MOVL C00694 V=800.0 PL=0
MOVL C00695 V=800.0 PL=0
MOVL C00696 V=800.0 PL=0
MOVL C00697 V=800.0 PL=0
MOVL C00698 V=800.0 PL=0
MOVL C00699 V=800.0 PL=0
MOVL C00700 V=800.0 PL=0
MOVL C00701 V=800.0 PL=0
MOVL C00702 V=800.0 PL=0
MOVL C00703 V=800.0 PL=0
MOVL C00704 V=800.0 PL=0
MOVL C00705 V=800.0 PL=0
MOVL C00706 V=800.0 PL=0
MOVL C00707 V=800.0 PL=0
MOVL C00708 V=800.0 PL=0
MOVL C00709 V=800.0 PL=0
MOVL C00710 V=800.0 PL=0
MOVL C00711 V=800.0 PL=0
MOVL C00712 V=800.0 PL=0
MOVL C00713 V=800.0 PL=0
MOVL C00714 V=800.0 PL=0
MOVL C00715 V=800.0 PL=0
MOVL C00716 V=800.0 PL=0
MOVL C00717 V=800.0 PL=0
MOVL C00718 V=800.0 PL=0
MOVL C00719 V=800.0 PL=0
MOVL C00720 V=800.0 PL=0
MOVL C00721 V=800.0 PL=0
MOVL C00722 V=800.0 PL=0
MOVL C00723 V=800.0 PL=0
MOVL C00724 V=800.0 PL=0
MOVL C00725 V=800.0 PL=0
MOVL C00726 V=800.0 PL=0
MOVL C00727 V=800.0 PL=0
MOVL C00728 V=800.0 PL=0
MOVL C00729 V=800.0 PL=0
MOVL C00730 V=800.0 PL=0
MOVL C00731 V=800.0 PL=0
MOVL C00732 V=800.0 PL=0
MOVL C00733 V=800.0 PL=0
MOVL C00734 V=800.0 PL=0
MOVL C00735 V=800.0 PL=0
MOVL C00736 V=800.0 PL=0
MOVL C00737 V=800.0 PL=0
MOVL C00738 V=800.0 PL=0
MOVL C00739 V=800.0 PL=0
MOVL C00740 V=800.0 PL=0
MOVL C00741 V=800.0 PL=0
MOVL C00742 V=800.0 PL=0
MOVL C00743 V=800.0 PL=0
MOVL C00744 V=800.0 PL=0
MOVL C00745 V=800.0 PL=0
MOVL C00746 V=800.0 PL=0
MOVL C00747 V=800.0 PL=0
MOVL C00748 V=800.0 PL=0
MOVL C00749 V=800.0 PL=0
MOVL C00750 V=800.0 PL=0
MOVL C00751 V=800.0 PL=0
MOVL C00752 V=800.0 PL=0
MOVL C00753 V=800.0 PL=0
MOVL C00754 V=800.0 PL=0
MOVL C00755 V=800.0 PL=0
MOVL C00756 V=800.0 PL=0
MOVL C00757 V=800.0 PL=0
MOVL C00758 V=800.0 PL=0
MOVL C00759 V=800.0 PL=0
MOVL C00760 V=800.0 PL=0
MOVL C00761 V=800.0 PL=0
MOVL C00762 V=800.0 PL=0
MOVL C00763 V=800.0 PL=0
MOVL C00764 V=800.0 PL=0
MOVL C00765 V=800.0 PL=0
MOVL C00766 V=800.0 PL=0
MOVL C00767 V=800.0 PL=0
MOVL C00768 V=800.0 PL=0
MOVL C00769 V=800.0 PL=0
MOVL C00770 V=800.0 PL=0
MOVL C00771 V=800.0 PL=0
MOVL C00772 V=800.0 PL=0
MOVL C00773 V=800.0 PL=0
MOVL C00774 V=800.0 PL=0
MOVL C00775 V=800.0 PL=0
MOVL C00776 V=800.0 PL=0
MOVL C00777 V=800.0 PL=0
MOVL C00778 V=800.0 PL=0
MOVL C00779 V=800.0 PL=0
MOVL C00780 V=800.0 PL=0
MOVL C00781 V=800.0 PL=0
MOVL C00782 V=800.0 PL=0
MOVL C00783 V=800.0 PL=0
MOVL C00784 V=800.0 PL=0
MOVL C00785 V=800.0 PL=0
MOVL C00786 V=800.0 PL=0
MOVL C00787 V=800.0 PL=0
MOVL C00788 V=800.0 PL=0
MOVL C00789 V=800.0 PL=0
MOVL C00790 V=800.0 PL=0
MOVL C00791 V=800.0 PL=0
MOVL C00792 V=800.0 PL=0
MOVL C00793 V=800.0 PL=0
MOVL C00794 V=800.0 PL=0
MOVL C00795 V=800.0 PL=0
MOVL C00796 V=800.0 PL=0
MOVL C00797 V=800.0 PL=0
MOVL C00798 V=800.0 PL=0
MOVL C00799 V=800.0 PL=0
MOVL C00800 V=800.0 PL=0
MOVL C00801 V=800.0 PL=0
MOVL C00802 V=800.0 PL=0
MOVL C00803 V=800.0 PL=0
MOVL C00804 V=800.0 PL=0
MOVL C00805 V=800.0 PL=0
MOVL C00806 V=800.0 PL=0
MOVL C00807 V=800.0 PL=0
MOVL C00808 V=800.0 PL=0
MOVL C00809 V=800.0 PL=0
MOVL C00810 V=800.0 PL=0
MOVL C00811 V=800.0 PL=0
MOVL C00812 V=800.0 PL=0
MOVL C00813 V=800.0 PL=0
MOVL C00814 V=800.0 PL=0
MOVL C00815 V=800.0 PL=0
MOVL C00816 V=800.0 PL=0
MOVL C00817 V=800.0 PL=0
MOVL C00818 V=800.0 PL=0
MOVL C00819 V=800.0 PL=0
MOVL C00820 V=800.0 PL=0
MOVL C00821 V=800.0 PL=0
MOVL C00822 V=800.0 PL=0
MOVL C00823 V=800.0 PL=0
MOVL C00824 V=800.0 PL=0
MOVL C00825 V=800.0 PL=0
MOVL C00826 V=800.0 PL=0
MOVL C00827 V=800.0 PL=0
MOVL C00828 V=800.0 PL=0
MOVL C00829 V=800.0 PL=0
MOVL C00830 V=800.0 PL=0
MOVL C00831 V=800.0 PL=0
MOVL C00832 V=800.0 PL=0
MOVL C00833 V=800.0 PL=0
MOVL C00834 V=800.0 PL=0
MOVL C00835 V=800.0 PL=0
MOVL C00836 V=800.0 PL=0
MOVL C00837 V=800.0 PL=0
MOVL C00838 V=800.0 PL=0
MOVL C00839 V=800.0 PL=0
MOVL C00840 V=800.0 PL=0
MOVL C00841 V=800.0 PL=0
MOVL C00842 V=800.0 PL=0
MOVL C00843 V=800.0 PL=0
MOVL C00844 V=800.0 PL=0
MOVL C00845 V=800.0 PL=0
MOVL C00846 V=800.0 PL=0
MOVL C00847 V=800.0 PL=0
MOVL C00848 V=800.0 PL=0
MOVL C00849 V=800.0 PL=0
MOVL C00850 V=800.0 PL=0
MOVL C00851 V=800.0 PL=0
MOVL C00852 V=800.0 PL=0
MOVL C00853 V=800.0 PL=0
MOVL C00854 V=800.0 PL=0
MOVL C00855 V=800.0 PL=0
MOVL C00856 V=800.0 PL=0
MOVL C00857 V=800.0 PL=0
MOVL C00858 V=800.0 PL=0
MOVL C00859 V=800.0 PL=0
MOVL C00860 V=800.0 PL=0
MOVL C00861 V=800.0 PL=0
MOVL C00862 V=800.0 PL=0
MOVL C00863 V=800.0 PL=0
MOVL C00864 V=800.0 PL=0
MOVL C00865 V=800.0 PL=0
MOVL C00866 V=800.0 PL=0
MOVL C00867 V=800.0 PL=0
MOVL C00868 V=800.0 PL=0
MOVL C00869 V=800.0 PL=0
MOVL C00870 V=800.0 PL=0
MOVL C00871 V=800.0 PL=0
MOVL C00872 V=800.0 PL=0
MOVL C00873 V=800.0 PL=0
MOVL C00874 V=800.0 PL=0
MOVL C00875 V=800.0 PL=0
MOVL C00876 V=800.0 PL=0
MOVL C00877 V=800.0 PL=0
MOVL C00878 V=800.0 PL=0
MOVL C00879 V=800.0 PL=0
MOVL C00880 V=800.0 PL=0
MOVL C00881 V=800.0 PL=0
MOVL C00882 V=800.0 PL=0
MOVL C00883 V=800.0 PL=0
MOVL C00884 V=800.0 PL=0
MOVL C00885 V=800.0 PL=0
MOVL C00886 V=800.0 PL=0
MOVL C00887 V=800.0 PL=0
MOVL C00888 V=800.0 PL=0
MOVL C00889 V=800.0 PL=0
MOVL C00890 V=800.0 PL=0
MOVL C00891 V=800.0 PL=0
MOVL C00892 V=800.0 PL=0
MOVL C00893 V=800.0 PL=0
MOVL C00894 V=800.0 PL=0
MOVL C00895 V=800.0 PL=0
MOVL C00896 V=800.0 PL=0
MOVL C00897 V=800.0 PL=0
MOVL C00898 V=800.0 PL=0
MOVL C00899 V=800.0 PL=0
MOVL C00900 V=800.0 PL=0
MOVL C00901 V=800.0 PL=0
MOVL C00902 V=800.0 PL=0
MOVL C00903 V=800.0 PL=0
MOVL C00904 V=800.0 PL=0
MOVL C00905 V=800.0 PL=0
MOVL C00906 V=800.0 PL=0
MOVL C00907 V=800.0 PL=0
MOVL C00908 V=800.0 PL=0
MOVL C00909 V=800.0 PL=0
MOVL C00910 V=800.0 PL=0
MOVL C00911 V=800.0 PL=0
MOVL C00912 V=800.0 PL=0
MOVL C00913 V=800.0 PL=0
MOVL C00914 V=800.0 PL=0
MOVL C00915 V=800.0 PL=0
MOVL C00916 V=800.0 PL=0
MOVL C00917 V=800.0 PL=0
MOVL C00918 V=800.0 PL=0
MOVL C00919 V=800.0 PL=0
MOVL C00920 V=800.0 PL=0
MOVL C00921 V=800.0 PL=0
MOVL C00922 V=800.0 PL=0
MOVL C00923 V=800.0 PL=0
MOVL C00924 V=800.0 PL=0
MOVL C00925 V=800.0 PL=0
MOVL C00926 V=800.0 PL=0
MOVL C00927 V=800.0 PL=0
MOVL C00928 V=800.0 PL=0
MOVL C00929 V=800.0 PL=0
MOVL C00930 V=800.0 PL=0
MOVL C00931 V=800.0 PL=0
MOVL C00932 V=800.0 PL=0
MOVL C00933 V=800.0 PL=0
MOVL C00934 V=800.0 PL=0
MOVL C00935 V=800.0 PL=0
MOVL C00936 V=800.0 PL=0
MOVL C00937 V=800.0 PL=0
MOVL C00938 V=800.0 PL=0
MOVL C00939 V=800.0 PL=0
MOVL C00940 V=800.0 PL=0
MOVL C00941 V=800.0 PL=0
MOVL C00942 V=800.0 PL=0
MOVL C00943 V=800.0 PL=0
MOVL C00944 V=800.0 PL=0
MOVL C00945 V=800.0 PL=0
MOVL C00946 V=800.0 PL=0
MOVL C00947 V=800.0 PL=0
MOVL C00948 V=800.0 PL=0
MOVL C00949 V=800.0 PL=0
MOVL C00950 V=800.0 PL=0
MOVL C00951 V=800.0 PL=0
MOVL C00952 V=800.0 PL=0
MOVL C00953 V=800.0 PL=0
MOVL C00954 V=800.0 PL=0
MOVL C00955 V=800.0 PL=0
MOVL C00956 V=800.0 PL=0
MOVL C00957 V=800.0 PL=0
MOVL C00958 V=800.0 PL=0
MOVL C00959 V=800.0 PL=0
MOVL C00960 V=800.0 PL=0
MOVL C00961 V=800.0 PL=0
MOVL C00962 V=800.0 PL=0
MOVL C00963 V=800.0 PL=0
MOVL C00964 V=800.0 PL=0
MOVL C00965 V=800.0 PL=0
MOVL C00966 V=800.0 PL=0
MOVL C00967 V=800.0 PL=0
MOVL C00968 V=800.0 PL=0
MOVL C00969 V=800.0 PL=0
MOVL C00970 V=800.0 PL=0
MOVL C00971 V=800.0 PL=0
MOVL C00972 V=800.0 PL=0
MOVL C00973 V=800.0 PL=0
MOVL C00974 V=800.0 PL=0
MOVL C00975 V=800.0 PL=0
MOVL C00976 V=800.0 PL=0
MOVL C00977 V=800.0 PL=0
MOVL C00978 V=800.0 PL=0
MOVL C00979 V=800.0 PL=0
MOVL C00980 V=800.0 PL=0
MOVL C00981 V=800.0 PL=0
MOVL C00982 V=800.0 PL=0
MOVL C00983 V=800.0 PL=0
MOVL C00984 V=800.0 PL=0
MOVL C00985 V=800.0 PL=0
MOVL C00986 V=800.0 PL=0
MOVL C00987 V=800.0 PL=0
MOVL C00988 V=800.0 PL=0
MOVL C00989 V=800.0 PL=0
MOVL C00990 V=800.0 PL=0
MOVL C00991 V=800.0 PL=0
MOVL C00992 V=800.0 PL=0
MOVL C00993 V=800.0 PL=0
MOVL C00994 V=800.0 PL=0
MOVL C00995 V=800.0 PL=0
MOVL C00996 V=800.0 PL=0
MOVL C00997 V=800.0 PL=0
MOVL C00998 V=800.0 PL=0
MOVL C00999 V=800.0 PL=0
MOVL C01000 V=800.0 PL=0
MOVL C01001 V=800.0 PL=0
MOVL C01002 V=800.0 PL=0
MOVL C01003 V=800.0 PL=0
MOVL C01004 V=800.0 PL=0
MOVL C01005 V=800.0 PL=0
MOVL C01006 V=800.0 PL=0
MOVL C01007 V=800.0 PL=0
MOVL C01008 V=800.0 PL=0
MOVL C01009 V=800.0 PL=0
MOVL C01010 V=800.0 PL=0
MOVL C01011 V=800.0 PL=0
MOVL C01012 V=800.0 PL=0
MOVL C01013 V=800.0 PL=0
MOVL C01014 V=800.0 PL=0
MOVL C01015 V=800.0 PL=0
MOVL C01016 V=800.0 PL=0
MOVL C01017 V=800.0 PL=0
MOVL C01018 V=800.0 PL=0
MOVL C01019 V=800.0 PL=0
MOVL C01020 V=800.0 PL=0
MOVL C01021 V=800.0 PL=0
MOVL C01022 V=800.0 PL=0
MOVL C01023 V=800.0 PL=0
MOVL C01024 V=800.0 PL=0
MOVL C01025 V=800.0 PL=0
MOVL C01026 V=800.0 PL=0
MOVL C01027 V=800.0 PL=0
MOVL C01028 V=800.0 PL=0
MOVL C01029 V=800.0 PL=0
MOVL C01030 V=800.0 PL=0
MOVL C01031 V=800.0 PL=0
MOVL C01032 V=800.0 PL=0
MOVL C01033 V=800.0 PL=0
MOVL C01034 V=800.0 PL=0
MOVL C01035 V=800.0 PL=0
MOVL C01036 V=800.0 PL=0
MOVL C01037 V=800.0 PL=0
MOVL C01038 V=800.0 PL=0
MOVL C01039 V=800.0 PL=0
MOVL C01040 V=800.0 PL=0
MOVL C01041 V=800.0 PL=0
MOVL C01042 V=800.0 PL=0
MOVL C01043 V=800.0 PL=0
MOVL C01044 V=800.0 PL=0
MOVL C01045 V=800.0 PL=0
MOVL C01046 V=800.0 PL=0
MOVL C01047 V=800.0 PL=0
MOVL C01048 V=800.0 PL=0
MOVL C01049 V=800.0 PL=0
MOVL C01050 V=800.0 PL=0
MOVL C01051 V=800.0 PL=0
MOVL C01052 V=800.0 PL=0
MOVL C01053 V=800.0 PL=0
MOVL C01054 V=800.0 PL=0
MOVL C01055 V=800.0 PL=0
MOVL C01056 V=800.0 PL=0
MOVL C01057 V=800.0 PL=0
MOVL C01058 V=800.0 PL=0
MOVL C01059 V=800.0 PL=0
MOVL C01060 V=800.0 PL=0
MOVL C01061 V=800.0 PL=0
MOVL C01062 V=800.0 PL=0
MOVL C01063 V=800.0 PL=0
MOVL C01064 V=800.0 PL=0
MOVL C01065 V=800.0 PL=0
MOVL C01066 V=800.0 PL=0
MOVL C01067 V=800.0 PL=0
MOVL C01068 V=800.0 PL=0
MOVL C01069 V=800.0 PL=0
MOVL C01070 V=800.0 PL=0
MOVL C01071 V=800.0 PL=0
MOVL C01072 V=800.0 PL=0
MOVL C01073 V=800.0 PL=0
MOVL C01074 V=800.0 PL=0
MOVL C01075 V=800.0 PL=0
MOVL C01076 V=800.0 PL=0
MOVL C01077 V=800.0 PL=0
MOVL C01078 V=800.0 PL=0
MOVL C01079 V=800.0 PL=0
MOVL C01080 V=800.0 PL=0
MOVL C01081 V=800.0 PL=0
MOVL C01082 V=800.0 PL=0
MOVL C01083 V=800.0 PL=0
MOVL C01084 V=800.0 PL=0
MOVL C01085 V=800.0 PL=0
MOVL C01086 V=800.0 PL=0
MOVL C01087 V=800.0 PL=0
MOVL C01088 V=800.0 PL=0
MOVL C01089 V=800.0 PL=0
MOVL C01090 V=800.0 PL=0
MOVL C01091 V=800.0 PL=0
MOVL C01092 V=800.0 PL=0
MOVL C01093 V=800.0 PL=0
MOVL C01094 V=800.0 PL=0
MOVL C01095 V=800.0 PL=0
MOVL C01096 V=800.0 PL=0
MOVL C01097 V=800.0 PL=0
MOVL C01098 V=800.0 PL=0
MOVL C01099 V=800.0 PL=0
MOVL C01100 V=800.0 PL=0
MOVL C01101 V=800.0 PL=0
MOVL C01102 V=800.0 PL=0
MOVL C01103 V=800.0 PL=0
MOVL C01104 V=800.0 PL=0
MOVL C01105 V=800.0 PL=0
MOVL C01106 V=800.0 PL=0
MOVL C01107 V=800.0 PL=0
MOVL C01108 V=800.0 PL=0
MOVL C01109 V=800.0 PL=0
MOVL C01110 V=800.0 PL=0
MOVL C01111 V=800.0 PL=0
MOVL C01112 V=800.0 PL=0
MOVL C01113 V=800.0 PL=0
MOVL C01114 V=800.0 PL=0
MOVL C01115 V=800.0 PL=0
MOVL C01116 V=800.0 PL=0
MOVL C01117 V=800.0 PL=0
MOVL C01118 V=800.0 PL=0
MOVL C01119 V=800.0 PL=0
MOVL C01120 V=800.0 PL=0
MOVL C01121 V=800.0 PL=0
MOVL C01122 V=800.0 PL=0
MOVL C01123 V=800.0 PL=0
MOVL C01124 V=800.0 PL=0
MOVL C01125 V=800.0 PL=0
MOVL C01126 V=800.0 PL=0
MOVL C01127 V=800.0 PL=0
MOVL C01128 V=800.0 PL=0
MOVL C01129 V=800.0 PL=0
MOVL C01130 V=800.0 PL=0
MOVL C01131 V=800.0 PL=0
MOVL C01132 V=800.0 PL=0
MOVL C01133 V=800.0 PL=0
MOVL C01134 V=800.0 PL=0
MOVL C01135 V=800.0 PL=0
MOVL C01136 V=800.0 PL=0
MOVL C01137 V=800.0 PL=0
MOVL C01138 V=800.0 PL=0
MOVL C01139 V=800.0 PL=0
MOVL C01140 V=800.0 PL=0
MOVL C01141 V=800.0 PL=0
MOVL C01142 V=800.0 PL=0
MOVL C01143 V=800.0 PL=0
MOVL C01144 V=800.0 PL=0
MOVL C01145 V=800.0 PL=0
MOVL C01146 V=800.0 PL=0
MOVL C01147 V=800.0 PL=0
MOVL C01148 V=800.0 PL=0
MOVL C01149 V=800.0 PL=0
MOVL C01150 V=800.0 PL=0
MOVL C01151 V=800.0 PL=0
MOVL C01152 V=800.0 PL=0
MOVL C01153 V=800.0 PL=0
MOVL C01154 V=800.0 PL=0
MOVL C01155 V=800.0 PL=0
MOVL C01156 V=800.0 PL=0
MOVL C01157 V=800.0 PL=0
MOVL C01158 V=800.0 PL=0
MOVL C01159 V=800.0 PL=0
MOVL C01160 V=800.0 PL=0
MOVL C01161 V=800.0 PL=0
MOVL C01162 V=800.0 PL=0
MOVL C01163 V=800.0 PL=0
MOVL C01164 V=800.0 PL=0
MOVL C01165 V=800.0 PL=0
MOVL C01166 V=800.0 PL=0
MOVL C01167 V=800.0 PL=0
MOVL C01168 V=800.0 PL=0
MOVL C01169 V=800.0 PL=0
MOVL C01170 V=800.0 PL=0
MOVL C01171 V=800.0 PL=0
MOVL C01172 V=800.0 PL=0
MOVL C01173 V=800.0 PL=0
MOVL C01174 V=800.0 PL=0
MOVL C01175 V=800.0 PL=0
MOVL C01176 V=800.0 PL=0
MOVL C01177 V=800.0 PL=0
MOVL C01178 V=800.0 PL=0
MOVL C01179 V=800.0 PL=0
MOVL C01180 V=800.0 PL=0
MOVL C01181 V=800.0 PL=0
MOVL C01182 V=800.0 PL=0
MOVL C01183 V=800.0 PL=0
MOVL C01184 V=800.0 PL=0
MOVL C01185 V=800.0 PL=0
MOVL C01186 V=800.0 PL=0
MOVL C01187 V=800.0 PL=0
MOVL C01188 V=800.0 PL=0
MOVL C01189 V=800.0 PL=0
MOVL C01190 V=800.0 PL=0
MOVL C01191 V=800.0 PL=0
MOVL C01192 V=800.0 PL=0
MOVL C01193 V=800.0 PL=0
MOVL C01194 V=800.0 PL=0
MOVL C01195 V=800.0 PL=0
MOVL C01196 V=800.0 PL=0
MOVL C01197 V=800.0 PL=0
MOVL C01198 V=800.0 PL=0
MOVL C01199 V=800.0 PL=0
MOVL C01200 V=800.0 PL=0
MOVL C01201 V=800.0 PL=0
MOVL C01202 V=800.0 PL=0
MOVL C01203 V=800.0 PL=0
MOVL C01204 V=800.0 PL=0
MOVL C01205 V=800.0 PL=0
MOVL C01206 V=800.0 PL=0
MOVL C01207 V=800.0 PL=0
MOVL C01208 V=800.0 PL=0
MOVL C01209 V=800.0 PL=0
MOVL C01210 V=800.0 PL=0
MOVL C01211 V=800.0 PL=0
MOVL C01212 V=800.0 PL=0
MOVL C01213 V=800.0 PL=0
MOVL C01214 V=800.0 PL=0
MOVL C01215 V=800.0 PL=0
MOVL C01216 V=800.0 PL=0
MOVL C01217 V=800.0 PL=0
MOVL C01218 V=800.0 PL=0
MOVL C01219 V=800.0 PL=0
MOVL C01220 V=800.0 PL=0
MOVL C01221 V=800.0 PL=0
MOVL C01222 V=800.0 PL=0
MOVL C01223 V=800.0 PL=0
MOVL C01224 V=800.0 PL=0
MOVL C01225 V=800.0 PL=0
MOVL C01226 V=800.0 PL=0
MOVL C01227 V=800.0 PL=0
MOVL C01228 V=800.0 PL=0
MOVL C01229 V=800.0 PL=0
MOVL C01230 V=800.0 PL=0
MOVL C01231 V=800.0 PL=0
MOVL C01232 V=800.0 PL=0
MOVL C01233 V=800.0 PL=0
MOVL C01234 V=800.0 PL=0
MOVL C01235 V=800.0 PL=0
MOVL C01236 V=800.0 PL=0
MOVL C01237 V=800.0 PL=0
MOVL C01238 V=800.0 PL=0
MOVL C01239 V=800.0 PL=0
MOVL C01240 V=800.0 PL=0
MOVL C01241 V=800.0 PL=0
MOVL C01242 V=800.0 PL=0
MOVL C01243 V=800.0 PL=0
MOVL C01244 V=800.0 PL=0
MOVL C01245 V=800.0 PL=0
MOVL C01246 V=800.0 PL=0
MOVL C01247 V=800.0 PL=0
MOVL C01248 V=800.0 PL=0
MOVL C01249 V=800.0 PL=0
MOVL C01250 V=800.0 PL=0
MOVL C01251 V=800.0 PL=0
MOVL C01252 V=800.0 PL=0
MOVL C01253 V=800.0 PL=0
MOVL C01254 V=800.0 PL=0
MOVL C01255 V=800.0 PL=0
MOVL C01256 V=800.0 PL=0
MOVL C01257 V=800.0 PL=0
MOVL C01258 V=800.0 PL=0
MOVL C01259 V=800.0 PL=0
MOVL C01260 V=800.0 PL=0
MOVL C01261 V=800.0 PL=0
MOVL C01262 V=800.0 PL=0
MOVL C01263 V=800.0 PL=0
MOVL C01264 V=800.0 PL=0
MOVL C01265 V=800.0 PL=0
MOVL C01266 V=800.0 PL=0
MOVL C01267 V=800.0 PL=0
MOVL C01268 V=800.0 PL=0
MOVL C01269 V=800.0 PL=0
MOVL C01270 V=800.0 PL=0
MOVL C01271 V=800.0 PL=0
MOVL C01272 V=800.0 PL=0
MOVL C01273 V=800.0 PL=0
MOVL C01274 V=800.0 PL=0
MOVL C01275 V=800.0 PL=0
MOVL C01276 V=800.0 PL=0
MOVL C01277 V=800.0 PL=0
MOVL C01278 V=800.0 PL=0
MOVL C01279 V=800.0 PL=0
MOVL C01280 V=800.0 PL=0
MOVL C01281 V=800.0 PL=0
MOVL C01282 V=800.0 PL=0
MOVL C01283 V=800.0 PL=0
MOVL C01284 V=800.0 PL=0
MOVL C01285 V=800.0 PL=0
MOVL C01286 V=800.0 PL=0
MOVL C01287 V=800.0 PL=0
MOVL C01288 V=800.0 PL=0
MOVL C01289 V=800.0 PL=0
MOVL C01290 V=800.0 PL=0
MOVL C01291 V=800.0 PL=0
MOVL C01292 V=800.0 PL=0
MOVL C01293 V=800.0 PL=0
MOVL C01294 V=800.0 PL=0
MOVL C01295 V=800.0 PL=0
MOVL C01296 V=800.0 PL=0
MOVL C01297 V=800.0 PL=0
MOVL C01298 V=800.0 PL=0
MOVL C01299 V=800.0 PL=0
MOVL C01300 V=800.0 PL=0
MOVL C01301 V=800.0 PL=0
MOVL C01302 V=800.0 PL=0
MOVL C01303 V=800.0 PL=0
MOVL C01304 V=800.0 PL=0
MOVL C01305 V=800.0 PL=0
MOVL C01306 V=800.0 PL=0
MOVL C01307 V=800.0 PL=0
MOVL C01308 V=800.0 PL=0
MOVL C01309 V=800.0 PL=0
MOVL C01310 V=800.0 PL=0
MOVL C01311 V=800.0 PL=0
MOVL C01312 V=800.0 PL=0
MOVL C01313 V=800.0 PL=0
MOVL C01314 V=800.0 PL=0
MOVL C01315 V=800.0 PL=0
MOVL C01316 V=800.0 PL=0
MOVL C01317 V=800.0 PL=0
MOVL C01318 V=800.0 PL=0
MOVL C01319 V=800.0 PL=0
MOVL C01320 V=800.0 PL=0
MOVL C01321 V=800.0 PL=0
MOVL C01322 V=800.0 PL=0
MOVL C01323 V=800.0 PL=0
MOVL C01324 V=800.0 PL=0
MOVL C01325 V=800.0 PL=0
MOVL C01326 V=800.0 PL=0
MOVL C01327 V=800.0 PL=0
MOVL C01328 V=800.0 PL=0
MOVL C01329 V=800.0 PL=0
MOVL C01330 V=800.0 PL=0
MOVL C01331 V=800.0 PL=0
MOVL C01332 V=800.0 PL=0
MOVL C01333 V=800.0 PL=0
MOVL C01334 V=800.0 PL=0
MOVL C01335 V=800.0 PL=0
MOVL C01336 V=800.0 PL=0
MOVL C01337 V=800.0 PL=0
MOVL C01338 V=800.0 PL=0
MOVL C01339 V=800.0 PL=0
MOVL C01340 V=800.0 PL=0
MOVL C01341 V=800.0 PL=0
MOVL C01342 V=800.0 PL=0
MOVL C01343 V=800.0 PL=0
MOVL C01344 V=800.0 PL=0
MOVL C01345 V=800.0 PL=0
MOVL C01346 V=800.0 PL=0
MOVL C01347 V=800.0 PL=0
MOVL C01348 V=800.0 PL=0
MOVL C01349 V=800.0 PL=0
MOVL C01350 V=800.0 PL=0
MOVL C01351 V=800.0 PL=0
MOVL C01352 V=800.0 PL=0
MOVL C01353 V=800.0 PL=0
MOVL C01354 V=800.0 PL=0
MOVL C01355 V=800.0 PL=0
MOVL C01356 V=800.0 PL=0
MOVL C01357 V=800.0 PL=0
MOVL C01358 V=800.0 PL=0
MOVL C01359 V=800.0 PL=0
MOVL C01360 V=800.0 PL=0
MOVL C01361 V=800.0 PL=0
MOVL C01362 V=800.0 PL=0
MOVL C01363 V=800.0 PL=0
MOVL C01364 V=800.0 PL=0
MOVL C01365 V=800.0 PL=0
MOVL C01366 V=800.0 PL=0
MOVL C01367 V=800.0 PL=0
MOVL C01368 V=800.0 PL=0
MOVL C01369 V=800.0 PL=0
MOVL C01370 V=800.0 PL=0
MOVL C01371 V=800.0 PL=0
MOVL C01372 V=800.0 PL=0
MOVL C01373 V=800.0 PL=0
MOVL C01374 V=800.0 PL=0
MOVL C01375 V=800.0 PL=0
MOVL C01376 V=800.0 PL=0
MOVL C01377 V=800.0 PL=0
MOVL C01378 V=800.0 PL=0
MOVL C01379 V=800.0 PL=0
MOVL C01380 V=800.0 PL=0
MOVL C01381 V=800.0 PL=0
MOVL C01382 V=800.0 PL=0
MOVL C01383 V=800.0 PL=0
MOVL C01384 V=800.0 PL=0
MOVL C01385 V=800.0 PL=0
MOVL C01386 V=800.0 PL=0
MOVL C01387 V=800.0 PL=0
MOVL C01388 V=800.0 PL=0
MOVL C01389 V=800.0 PL=0
MOVL C01390 V=800.0 PL=0
MOVL C01391 V=800.0 PL=0
MOVL C01392 V=800.0 PL=0
MOVL C01393 V=800.0 PL=0
MOVL C01394 V=800.0 PL=0
MOVL C01395 V=800.0 PL=0
MOVL C01396 V=800.0 PL=0
MOVL C01397 V=800.0 PL=0
MOVL C01398 V=800.0 PL=0
MOVL C01399 V=800.0 PL=0
MOVL C01400 V=800.0 PL=0
MOVL C01401 V=800.0 PL=0
MOVL C01402 V=800.0 PL=0
MOVL C01403 V=800.0 PL=0
MOVL C01404 V=800.0 PL=0
MOVL C01405 V=800.0 PL=0
MOVL C01406 V=800.0 PL=0
MOVL C01407 V=800.0 PL=0
MOVL C01408 V=800.0 PL=0
MOVL C01409 V=800.0 PL=0
MOVL C01410 V=800.0 PL=0
MOVL C01411 V=800.0 PL=0
MOVL C01412 V=800.0 PL=0
MOVL C01413 V=800.0 PL=0
MOVL C01414 V=800.0 PL=0
MOVL C01415 V=800.0 PL=0
MOVL C01416 V=800.0 PL=0
MOVL C01417 V=800.0 PL=0
MOVL C01418 V=800.0 PL=0
MOVL C01419 V=800.0 PL=0
MOVL C01420 V=800.0 PL=0
MOVL C01421 V=800.0 PL=0
MOVL C01422 V=800.0 PL=0
MOVL C01423 V=800.0 PL=0
MOVL C01424 V=800.0 PL=0
MOVL C01425 V=800.0 PL=0
MOVL C01426 V=800.0 PL=0
MOVL C01427 V=800.0 PL=0
MOVL C01428 V=800.0 PL=0
MOVL C01429 V=800.0 PL=0
MOVL C01430 V=800.0 PL=0
MOVL C01431 V=800.0 PL=0
MOVL C01432 V=800.0 PL=0
MOVL C01433 V=800.0 PL=0
MOVL C01434 V=800.0 PL=0
MOVL C01435 V=800.0 PL=0
MOVL C01436 V=800.0 PL=0
MOVL C01437 V=800.0 PL=0
MOVL C01438 V=800.0 PL=0
MOVL C01439 V=800.0 PL=0
MOVL C01440 V=800.0 PL=0
MOVL C01441 V=800.0 PL=0
MOVL C01442 V=800.0 PL=0
MOVL C01443 V=800.0 PL=0
MOVL C01444 V=800.0 PL=0
MOVL C01445 V=800.0 PL=0
MOVL C01446 V=800.0 PL=0
MOVL C01447 V=800.0 PL=0
MOVL C01448 V=800.0 PL=0
MOVL C01449 V=800.0 PL=0
MOVL C01450 V=800.0 PL=0
MOVL C01451 V=800.0 PL=0
MOVL C01452 V=800.0 PL=0
MOVL C01453 V=800.0 PL=0
MOVL C01454 V=800.0 PL=0
MOVL C01455 V=800.0 PL=0
MOVL C01456 V=800.0 PL=0
MOVL C01457 V=800.0 PL=0
MOVL C01458 V=800.0 PL=0
MOVL C01459 V=800.0 PL=0
MOVL C01460 V=800.0 PL=0
MOVL C01461 V=800.0 PL=0
MOVL C01462 V=800.0 PL=0
MOVL C01463 V=800.0 PL=0
MOVL C01464 V=800.0 PL=0
MOVL C01465 V=800.0 PL=0
MOVL C01466 V=800.0 PL=0
MOVL C01467 V=800.0 PL=0
MOVL C01468 V=800.0 PL=0
MOVL C01469 V=800.0 PL=0
MOVL C01470 V=800.0 PL=0
MOVL C01471 V=800.0 PL=0
MOVL C01472 V=800.0 PL=0
MOVL C01473 V=800.0 PL=0
MOVL C01474 V=800.0 PL=0
MOVL C01475 V=800.0 PL=0
MOVL C01476 V=800.0 PL=0
MOVL C01477 V=800.0 PL=0
MOVL C01478 V=800.0 PL=0
MOVL C01479 V=800.0 PL=0
MOVL C01480 V=800.0 PL=0
MOVL C01481 V=800.0 PL=0
MOVL C01482 V=800.0 PL=0
MOVL C01483 V=800.0 PL=0
MOVL C01484 V=800.0 PL=0
MOVL C01485 V=800.0 PL=0
MOVL C01486 V=800.0 PL=0
MOVL C01487 V=800.0 PL=0
MOVL C01488 V=800.0 PL=0
MOVL C01489 V=800.0 PL=0
MOVL C01490 V=800.0 PL=0
MOVL C01491 V=800.0 PL=0
MOVL C01492 V=800.0 PL=0
MOVL C01493 V=800.0 PL=0
MOVL C01494 V=800.0 PL=0
MOVL C01495 V=800.0 PL=0
MOVL C01496 V=800.0 PL=0
MOVL C01497 V=800.0 PL=0
MOVL C01498 V=800.0 PL=0
MOVL C01499 V=800.0 PL=0
MOVL C01500 V=800.0 PL=0
MOVL C01501 V=800.0 PL=0
MOVL C01502 V=800.0 PL=0
MOVL C01503 V=800.0 PL=0
MOVL C01504 V=800.0 PL=0
MOVL C01505 V=800.0 PL=0
MOVL C01506 V=800.0 PL=0
MOVL C01507 V=800.0 PL=0
MOVL C01508 V=800.0 PL=0
MOVL C01509 V=800.0 PL=0
MOVL C01510 V=800.0 PL=0
MOVL C01511 V=800.0 PL=0
MOVL C01512 V=800.0 PL=0
MOVL C01513 V=800.0 PL=0
MOVL C01514 V=800.0 PL=0
MOVL C01515 V=800.0 PL=0
MOVL C01516 V=800.0 PL=0
MOVL C01517 V=800.0 PL=0
MOVL C01518 V=800.0 PL=0
MOVL C01519 V=800.0 PL=0
MOVL C01520 V=800.0 PL=0
MOVL C01521 V=800.0 PL=0
MOVL C01522 V=800.0 PL=0
MOVL C01523 V=800.0 PL=0
MOVL C01524 V=800.0 PL=0
MOVL C01525 V=800.0 PL=0
MOVL C01526 V=800.0 PL=0
MOVL C01527 V=800.0 PL=0
MOVL C01528 V=800.0 PL=0
MOVL C01529 V=800.0 PL=0
MOVL C01530 V=800.0 PL=0
MOVL C01531 V=800.0 PL=0
MOVL C01532 V=800.0 PL=0
MOVL C01533 V=800.0 PL=0
MOVL C01534 V=800.0 PL=0
MOVL C01535 V=800.0 PL=0
MOVL C01536 V=800.0 PL=0
MOVL C01537 V=800.0 PL=0
MOVL C01538 V=800.0 PL=0
MOVL C01539 V=800.0 PL=0
MOVL C01540 V=800.0 PL=0
MOVL C01541 V=800.0 PL=0
MOVL C01542 V=800.0 PL=0
MOVL C01543 V=800.0 PL=0
MOVL C01544 V=800.0 PL=0
MOVL C01545 V=800.0 PL=0
MOVL C01546 V=800.0 PL=0
MOVL C01547 V=800.0 PL=0
MOVL C01548 V=800.0 PL=0
MOVL C01549 V=800.0 PL=0
MOVL C01550 V=800.0 PL=0
MOVL C01551 V=800.0 PL=0
MOVL C01552 V=800.0 PL=0
MOVL C01553 V=800.0 PL=0
MOVL C01554 V=800.0 PL=0
MOVL C01555 V=800.0 PL=0
MOVL C01556 V=800.0 PL=0
MOVL C01557 V=800.0 PL=0
MOVL C01558 V=800.0 PL=0
MOVL C01559 V=800.0 PL=0
MOVL C01560 V=800.0 PL=0
MOVL C01561 V=800.0 PL=0
MOVL C01562 V=800.0 PL=0
MOVL C01563 V=800.0 PL=0
MOVL C01564 V=800.0 PL=0
MOVL C01565 V=800.0 PL=0
MOVL C01566 V=800.0 PL=0
MOVL C01567 V=800.0 PL=0
MOVL C01568 V=800.0 PL=0
MOVL C01569 V=800.0 PL=0
MOVL C01570 V=800.0 PL=0
MOVL C01571 V=800.0 PL=0
MOVL C01572 V=800.0 PL=0
MOVL C01573 V=800.0 PL=0
MOVL C01574 V=800.0 PL=0
MOVL C01575 V=800.0 PL=0
MOVL C01576 V=800.0 PL=0
MOVL C01577 V=800.0 PL=0
MOVL C01578 V=800.0 PL=0
MOVL C01579 V=800.0 PL=0
MOVL C01580 V=800.0 PL=0
MOVL C01581 V=800.0 PL=0
MOVL C01582 V=800.0 PL=0
MOVL C01583 V=800.0 PL=0
MOVL C01584 V=800.0 PL=0
MOVL C01585 V=800.0 PL=0
MOVL C01586 V=800.0 PL=0
MOVL C01587 V=800.0 PL=0
MOVL C01588 V=800.0 PL=0
MOVL C01589 V=800.0 PL=0
MOVL C01590 V=800.0 PL=0
MOVL C01591 V=800.0 PL=0
MOVL C01592 V=800.0 PL=0
MOVL C01593 V=800.0 PL=0
MOVL C01594 V=800.0 PL=0
MOVL C01595 V=800.0 PL=0
MOVL C01596 V=800.0 PL=0
MOVL C01597 V=800.0 PL=0
MOVL C01598 V=800.0 PL=0
MOVL C01599 V=800.0 PL=0
MOVL C01600 V=800.0 PL=0
MOVL C01601 V=800.0 PL=0
MOVL C01602 V=800.0 PL=0
MOVL C01603 V=800.0 PL=0
MOVL C01604 V=800.0 PL=0
MOVL C01605 V=800.0 PL=0
MOVL C01606 V=800.0 PL=0
MOVL C01607 V=800.0 PL=0
MOVL C01608 V=800.0 PL=0
MOVL C01609 V=800.0 PL=0
MOVL C01610 V=800.0 PL=0
MOVL C01611 V=800.0 PL=0
MOVL C01612 V=800.0 PL=0
MOVL C01613 V=800.0 PL=0
MOVL C01614 V=800.0 PL=0
MOVL C01615 V=800.0 PL=0
MOVL C01616 V=800.0 PL=0
MOVL C01617 V=800.0 PL=0
MOVL C01618 V=800.0 PL=0
MOVL C01619 V=800.0 PL=0
MOVL C01620 V=800.0 PL=0
MOVL C01621 V=800.0 PL=0
MOVL C01622 V=800.0 PL=0
MOVL C01623 V=800.0 PL=0
MOVL C01624 V=800.0 PL=0
MOVL C01625 V=800.0 PL=0
MOVL C01626 V=800.0 PL=0
MOVL C01627 V=800.0 PL=0
MOVL C01628 V=800.0 PL=0
MOVL C01629 V=800.0 PL=0
MOVL C01630 V=800.0 PL=0
MOVL C01631 V=800.0 PL=0
MOVL C01632 V=800.0 PL=0
MOVL C01633 V=800.0 PL=0
MOVL C01634 V=800.0 PL=0
MOVL C01635 V=800.0 PL=0
MOVL C01636 V=800.0 PL=0
MOVL C01637 V=800.0 PL=0
MOVL C01638 V=800.0 PL=0
MOVL C01639 V=800.0 PL=0
MOVL C01640 V=800.0 PL=0
MOVL C01641 V=800.0 PL=0
MOVL C01642 V=800.0 PL=0
MOVL C01643 V=800.0 PL=0
MOVL C01644 V=800.0 PL=0
MOVL C01645 V=800.0 PL=0
MOVL C01646 V=800.0 PL=0
MOVL C01647 V=800.0 PL=0
MOVL C01648 V=800.0 PL=0
MOVL C01649 V=800.0 PL=0
MOVL C01650 V=800.0 PL=0
MOVL C01651 V=800.0 PL=0
MOVL C01652 V=800.0 PL=0
MOVL C01653 V=800.0 PL=0
MOVL C01654 V=800.0 PL=0
MOVL C01655 V=800.0 PL=0
MOVL C01656 V=800.0 PL=0
MOVL C01657 V=800.0 PL=0
MOVL C01658 V=800.0 PL=0
MOVL C01659 V=800.0 PL=0
MOVL C01660 V=800.0 PL=0
MOVL C01661 V=800.0 PL=0
MOVL C01662 V=800.0 PL=0
MOVL C01663 V=800.0 PL=0
MOVL C01664 V=800.0 PL=0
MOVL C01665 V=800.0 PL=0
MOVL C01666 V=800.0 PL=0
MOVL C01667 V=800.0 PL=0
MOVL C01668 V=800.0 PL=0
MOVL C01669 V=800.0 PL=0
MOVL C01670 V=800.0 PL=0
MOVL C01671 V=800.0 PL=0
MOVL C01672 V=800.0 PL=0
MOVL C01673 V=800.0 PL=0
MOVL C01674 V=800.0 PL=0
MOVL C01675 V=800.0 PL=0
MOVL C01676 V=800.0 PL=0
MOVL C01677 V=800.0 PL=0
MOVL C01678 V=800.0 PL=0
MOVL C01679 V=800.0 PL=0
MOVL C01680 V=800.0 PL=0
MOVL C01681 V=800.0 PL=0
MOVL C01682 V=800.0 PL=0
MOVL C01683 V=800.0 PL=0
MOVL C01684 V=800.0 PL=0
MOVL C01685 V=800.0 PL=0
MOVL C01686 V=800.0 PL=0
MOVL C01687 V=800.0 PL=0
MOVL C01688 V=800.0 PL=0
MOVL C01689 V=800.0 PL=0
